	(* --- Visu controler --- *)
	iMAX_AXIS_FRAMES						: USINT := 20;														(* Maximum frames of displayed axis in manual mode *)
	iMAX_CYLINDER_FRAMES					: USINT := 42;														(* Maximum frames of displayed cylinders in manual mode *)
	iMAX_OUTPUT_FRAMES						: USINT := 144;														(* Maximum frames of displayed outputs in manual mode *)
	iMAX_INPUT_FRAMES						: USINT := 144;														(* Maximum frames of displayed inputs in manual mode *)
	iMAX_SAFE_INPUT_FRAMES					: USINT := 36;														(* Maximum frames of displayed safe inputs in manual mode *)
	iMAX_SAFE_OUTPUT_FRAMES					: USINT := 36;														(* Maximum frames of displayed safe outputs in manual mode *)
	iMAX_ROBOT_FRAMES						: USINT := 10;														(* Maximum frames of displayed safe outputs in manual mode *)
	                                                        													
	iAXIS_PER_PAGE							: USINT := 2;														(* Number of axis displayed on single page *)
	iCYLINDERS_PER_PAGE						: USINT := 3;														(* Number of cylinders dislayed on single page *)
	iOUTPUTS_PER_PAGE						: USINT := 12;														(* Number of outputs displayed on single page *)
	iINPUTS_PER_PAGE						: USINT := 12;														(* Number of inputs displayed on single page *)
	iSAFE_INPUTS_PER_PAGE					: USINT := 6;														(* Number of safe inputs displayed on single page*)
	iSAFE_OUTPUTS_PER_PAGE					: USINT := 6;														(* Number of safe outputs displayed on single page *)
	iRECIPE_PARAMETERS_PER_PAGE				: USINT := 8;														(* Number of recipes parameters displayed on single page *)
	iROBOTS_PER_PAGE						: USINT := 1;														(* Number of recipes parameters displayed on single page *)
	
	iMAX_AXIS_PAGES							: USINT := iMAX_AXIS_FRAMES / iAXIS_PER_PAGE;						(* Defines maximum pages of axis HMI frames in manual mode *)
	iMAX_CYLINDER_PAGES						: USINT := iMAX_CYLINDER_FRAMES / iCYLINDERS_PER_PAGE;				(* Defines maximum pages of cylinders HMI frames in manual mode *)
	iMAX_OUTPUT_PAGES						: USINT := iMAX_OUTPUT_FRAMES / iOUTPUTS_PER_PAGE;					(* Defines maximum pages of digital outputs HMI frames in manual mode *)
	iMAX_INPUT_PAGES						: USINT := iMAX_INPUT_FRAMES / iINPUTS_PER_PAGE;					(* Defines maximum pages of digital inputs HMI frames in manual mode *)
	iMAX_SAFE_INPUT_PAGES					: USINT := iMAX_SAFE_INPUT_FRAMES / iSAFE_INPUTS_PER_PAGE;			(* Defines maximum pages of safe inputs HMI frames in manual mode *)
	iMAX_SAFE_OUTPUT_PAGES					: USINT := iMAX_SAFE_OUTPUT_FRAMES / iSAFE_OUTPUTS_PER_PAGE;		(* Defines maximum pages of safe outputs HMI frames in manual mode *)
	iMAX_RECIPES_PAGES						: USINT := iMAX_NUMBER_OF_RECIPES / iRECIPE_PARAMETERS_PER_PAGE;	(* Defines maximum pages of recipes parameter HMI frames in manual mode *)
	iMAX_ROBOT_PAGES						: USINT := iMAX_ROBOT_FRAMES / iROBOTS_PER_PAGE;					(* Defines maximum pages of robots HMI frames *)

	(* --- CSV Data Exchanger --- *)
	iMAX_CSV_ROWS 							: UDINT := 100;
	iMAX_CSV_COLUMNS 						: UDINT := 8;
	iMAX_CSV_FIELD_LENGTH					: UDINT := 100;
END_VAR
VAR_GLOBAL
	(* --- Machine data ---*)
	sMACHINE_NAME							: STRING := 'PSE Shell Test Machine';								(* Full machine project name *)
	sSOFTWARE_VERSION						: STRING := '1.0.1.0';												(* Last taged version of control software *)
	
	(* --- Shell common features ---*)
	fbMachineTime							: FB_LocalSystemTime; 												(* Main machine clock - used by implementation of other utilites like Logger and Alarm Controler *)
	fbMachineLogger 						: FB_FileLogger; 													(* Main machine logger - registers everything that happens on machine *)

	(* --- Shell Machine ---*)
	stShell : ST_Shell;	(* This structure contains references to Shell modules, recipe parameters and auxilary bit flags *)
END_VAR

// ---- POUs/Libs/0_Checks/GVL_Checks.TcGVL
{attribute 'qualified_only'}
VAR_GLOBAL PERSISTENT
	dCheckBounds					: DINT;			// Licznik przekroczen zakresu indexow, np. tablic
	dCheckDivDInt					: DINT;			// Licznik prob dzielenia Dint przez 0
	dCheckDivLInt					: DINT; 		// Licznik prob dzielenia LInt przez 0
	dCheckDivLReal					: DINT; 		// Licznik prob dzielenia LREAL przez 0
	dCheckDivReal					: DINT; 		// Licznik prob dzielenia REAL przez 0
	dCheckRangeSigned				: DINT;			// Licznik przekroczen liczby znakowej
	dCheckRangeUnsigned				: DINT; 		// Licznik przekroczen liczby bezznakowej
END_VAR

// ---- POUs/Libs/Alarms/AlarmControler/I_AlarmControler.TcIO
INTERFACE I_AlarmControler

PROPERTY Active : REFERENCE TO BOOL
GET
END_GET
END_PROPERTY

PROPERTY ActiveCritical : REFERENCE TO UDINT
GET
END_GET
END_PROPERTY

PROPERTY ActiveError : REFERENCE TO UDINT
GET
END_GET
END_PROPERTY

PROPERTY ActiveInfo : REFERENCE TO UDINT
GET
END_GET
END_PROPERTY

PROPERTY ActiveVerbose : REFERENCE TO UDINT
GET
END_GET
END_PROPERTY

PROPERTY ActiveWarrning : REFERENCE TO UDINT
GET
END_GET
END_PROPERTY

PROPERTY Busy : REFERENCE TO BOOL
GET
END_GET
END_PROPERTY

PROPERTY Error : REFERENCE TO BOOL
GET
END_GET
END_PROPERTY

PROPERTY FileName : STRING
GET
END_GET
SET
END_SET
END_PROPERTY

PROPERTY MaxEvents : UDINT
GET
END_GET
END_PROPERTY

METHOD MR_Abort : BOOL
VAR_INPUT
END_VAR
END_METHOD

METHOD MR_Clear : BOOL
VAR_INPUT
	ipFilter : I_TcEventFilter;
	bResetConfirmation : BOOL;
END_VAR
END_METHOD

METHOD MR_ClearAll : BOOL
VAR_INPUT
	bResetConfirmation : BOOL;
END_VAR
END_METHOD

METHOD MR_Confirm : BOOL
VAR_INPUT
	ipFilter : I_TcEventFilter;
END_VAR
END_METHOD

METHOD MR_ConfirmAll : BOOL
VAR_INPUT
	bResetConfirmation : BOOL;
END_VAR
END_METHOD

METHOD MR_Export : BOOL
VAR_INPUT
END_VAR
END_METHOD

METHOD MR_FirstCycle : BOOL
VAR_INPUT
	sName 		: STRING;
	sFileName 	: STRING;
END_VAR
END_METHOD

METHOD MR_Init : BOOL
VAR_INPUT
END_VAR
END_METHOD

PROPERTY Name : REFERENCE TO STRING
GET
END_GET
END_PROPERTY

PROPERTY State : REFERENCE TO E_AlarmControlerState
GET
END_GET
END_PROPERTY

END_INTERFACE

// ---- POUs/Libs/Axis/I_UniversalAxis.TcIO
INTERFACE I_UniversalAxis

PROPERTY Acceleration : LREAL
GET
END_GET
SET
END_SET
END_PROPERTY

PROPERTY Active : REFERENCE TO BOOL
GET
END_GET
END_PROPERTY

PROPERTY ActualPosition : REFERENCE TO LREAL
GET
END_GET
END_PROPERTY

PROPERTY ActualVelocity : REFERENCE TO LREAL
GET
END_GET
END_PROPERTY

PROPERTY AxisErrorID : REFERENCE TO UDINT
GET
END_GET
END_PROPERTY

PROPERTY AxisRef : AXIS_REF
GET
END_GET
SET
END_SET
END_PROPERTY

PROPERTY BufferMode : MC_BufferMode
GET
END_GET
SET
END_SET
END_PROPERTY

PROPERTY Busy : REFERENCE TO BOOL
GET
END_GET
END_PROPERTY

PROPERTY Deceleration : LREAL
GET
END_GET
SET
END_SET
END_PROPERTY

PROPERTY Direction : Tc2_MC2.MC_Direction
GET
END_GET
SET
END_SET
END_PROPERTY

PROPERTY Error : REFERENCE TO BOOL
GET
END_GET
END_PROPERTY

PROPERTY ErrorID : REFERENCE TO UDINT
GET
END_GET
END_PROPERTY

PROPERTY Halted : REFERENCE TO BOOL
GET
END_GET
END_PROPERTY

PROPERTY InPosition : REFERENCE TO BOOL
GET
END_GET
END_PROPERTY

PROPERTY InVelocity : REFERENCE TO BOOL
GET
END_GET
END_PROPERTY

PROPERTY IsHomed : REFERENCE TO BOOL
GET
END_GET
END_PROPERTY

PROPERTY Jerk : LREAL
GET
END_GET
SET
END_SET
END_PROPERTY

PROPERTY JogAcceleration : LREAL
GET
END_GET
SET
END_SET
END_PROPERTY

PROPERTY JogDeceleration : LREAL
GET
END_GET
SET
END_SET
END_PROPERTY

PROPERTY JogDirection : E_AxisJogDirection
GET
END_GET
SET
END_SET
END_PROPERTY

PROPERTY JogDone : REFERENCE TO BOOL
GET
END_GET
END_PROPERTY

PROPERTY JogJerk : LREAL
GET
END_GET
SET
END_SET
END_PROPERTY

PROPERTY JogMode : E_JogMode
GET
END_GET
SET
END_SET
END_PROPERTY

PROPERTY JogPosition : LREAL
GET
END_GET
SET
END_SET
END_PROPERTY

PROPERTY JogVelocity : LREAL
GET
END_GET
SET
END_SET
END_PROPERTY

PROPERTY LagError : LREAL
GET
END_GET
END_PROPERTY

PROPERTY MoveActive : REFERENCE TO BOOL
GET
END_GET
END_PROPERTY

METHOD MR_Abort : BOOL
END_METHOD

METHOD MR_FirstCycle
VAR_INPUT
	sName 				: STRING; 	(* Axis object name *)
	sMeasurementUnits	: STRING;	(* Measurement units used by axis *)
	bModulo				: BOOL;		(* Axis is periodic *)
END_VAR
END_METHOD

METHOD MR_Halt : BOOL
END_METHOD

METHOD MR_Home : BOOL
VAR_INPUT
	lrHomePosition : LREAL;
END_VAR
END_METHOD

METHOD MR_Init : BOOL
END_METHOD

METHOD MR_Jog : BOOL
VAR_INPUT
	//lrJogPosition : LREAL;
	//eJogDirection : E_AxisJogDirection;
	//eJogMode	  : E_JogMode;
	bJogActive	  : BOOL;
END_VAR
END_METHOD

METHOD MR_MoveAbsolute : BOOL
VAR_INPUT
	lrAbsolutePosition : LREAL;
END_VAR
END_METHOD

METHOD MR_MoveAdditive : BOOL
VAR_INPUT
	lrRelativeDistance : LREAL;
END_VAR
END_METHOD

METHOD MR_MoveRelative : BOOL
VAR_INPUT
	lrRelativeDistance : LREAL;
END_VAR
END_METHOD

METHOD MR_MoveVelocity : BOOL
END_METHOD

METHOD MR_Reset : BOOL
END_METHOD

METHOD MR_Stop : BOOL
END_METHOD

PROPERTY Name : STRING
GET
END_GET
SET
END_SET
END_PROPERTY

PROPERTY Options : ST_MoveOptions
GET
END_GET
SET
END_SET
END_PROPERTY

PROPERTY Override : LREAL
GET
END_GET
SET
END_SET
END_PROPERTY

PROPERTY PowerOn : REFERENCE TO BOOL
GET
END_GET
END_PROPERTY

PROPERTY SetpointPosition : LREAL
GET
END_GET
END_PROPERTY

PROPERTY SetpointVelocity : LREAL
GET
END_GET
END_PROPERTY

PROPERTY State : REFERENCE TO E_AxisState
GET
END_GET
END_PROPERTY

PROPERTY StatePlcOpen : REFERENCE TO E_AxisStatePlcOpen
GET
END_GET
END_PROPERTY

PROPERTY StopDeceleration : LREAL
GET
END_GET
SET
END_SET
END_PROPERTY

PROPERTY StopJerk : LREAL
GET
END_GET
SET
END_SET
END_PROPERTY

PROPERTY Stopped : REFERENCE TO BOOL
GET
END_GET
END_PROPERTY

PROPERTY Unit : STRING
GET
END_GET
SET
END_SET
END_PROPERTY

PROPERTY Velocity : LREAL
GET
END_GET
SET
END_SET
END_PROPERTY

END_INTERFACE

// ---- POUs/Libs/Communication/TcpIp/Tcp Device/I_TcpDevice.TcIO
INTERFACE I_TcpDevice

PROPERTY Active : REFERENCE TO BOOL
GET
END_GET
END_PROPERTY

PROPERTY AmsNetId : T_IPv4Addr
GET
END_GET
SET
END_SET
END_PROPERTY

PROPERTY Error : REFERENCE TO BOOL
GET
END_GET
END_PROPERTY

PROPERTY ErrorID : REFERENCE TO UDINT
GET
END_GET
END_PROPERTY

PROPERTY Host : T_IPv4Addr
GET
END_GET
SET
END_SET
END_PROPERTY

PROPERTY LastRecivedMessage : ST_TcpBufferData
GET
END_GET
END_PROPERTY

METHOD MR_Abort : BOOL
VAR_INPUT
END_VAR
END_METHOD

METHOD MR_FirstCycle : BOOL
VAR_INPUT
	sName 		: STRING;		(*  *)
	sHost		: T_IPv4Addr;	(*  *)
	sAmsNetID	: T_AmsNetID;	(*  *)
	iPort		: UINT;			(*  *)
	tTimeout	: TIME;			(*  *)
END_VAR
END_METHOD

METHOD MR_Init : BOOL
VAR_INPUT
END_VAR
END_METHOD

PROPERTY NextRecivedMessage : ST_TcpBufferData
GET
END_GET
END_PROPERTY

PROPERTY Port : UINT
GET
END_GET
SET
END_SET
END_PROPERTY

PROPERTY State : REFERENCE TO E_TcpIpDeviceState
GET
END_GET
END_PROPERTY

PROPERTY Timeout : TIME
GET
END_GET
SET
END_SET
END_PROPERTY

END_INTERFACE

// ---- POUs/Libs/Cylinder/Universal Cylinder/I_UniversalCylinder.TcIO
INTERFACE I_UniversalCylinder

PROPERTY Active : REFERENCE TO BOOL
GET
END_GET
END_PROPERTY

PROPERTY ActiveTimeout : TIME
GET
END_GET
SET
END_SET
END_PROPERTY

PROPERTY Busy : REFERENCE TO BOOL
GET
END_GET
END_PROPERTY

PROPERTY Delay : TIME
GET
END_GET
SET
END_SET
END_PROPERTY

PROPERTY Error : REFERENCE TO BOOL
GET
END_GET
END_PROPERTY

PROPERTY ErrorID : REFERENCE TO E_CylinderError
GET
END_GET
END_PROPERTY

PROPERTY HomeTimeout : TIME
GET
END_GET
SET
END_SET
END_PROPERTY

PROPERTY MoveActiveTime : REFERENCE TO TIME
GET
END_GET
END_PROPERTY

PROPERTY MoveHomeTime : REFERENCE TO TIME
GET
END_GET
END_PROPERTY

METHOD MR_Abort : BOOL
VAR_INPUT
END_VAR
END_METHOD

METHOD MR_FirstCycle : BOOL
VAR_INPUT
sName 							: STRING;
	sHomeSensorModuleType			: STRING;
	sHomeSensorPortID				: STRING;
	sActiveSensorModuleType			: STRING;
	sActiveSensorPortID				: STRING;
	tGoHomeTimeout					: TIME;
	tGoActiveTimeout				: TIME;
	tDelay							: TIME;
END_VAR
END_METHOD

METHOD MR_GoActive : BOOL
VAR_INPUT
END_VAR
END_METHOD

METHOD MR_GoHome : BOOL
VAR_INPUT
END_VAR
END_METHOD

METHOD MR_Init : BOOL
VAR_INPUT
END_VAR
END_METHOD

METHOD MR_Release : BOOL
VAR_INPUT
END_VAR
END_METHOD

METHOD MR_Reset : BOOL
VAR_INPUT
END_VAR
END_METHOD

PROPERTY Name : STRING
GET
END_GET
SET
END_SET
END_PROPERTY

PROPERTY PositionActive : REFERENCE TO BOOL
GET
END_GET
END_PROPERTY

PROPERTY PositionHold : REFERENCE TO BOOL
GET
END_GET
END_PROPERTY

PROPERTY PositionHome : REFERENCE TO BOOL
GET
END_GET
END_PROPERTY

PROPERTY Simulation : BOOL
GET
END_GET
SET
END_SET
END_PROPERTY

PROPERTY State : REFERENCE TO E_CylinderState
GET
END_GET
END_PROPERTY

END_INTERFACE

// ---- POUs/Libs/Digital Devices/Digital Device/I_DigitalDevice.TcIO
INTERFACE I_DigitalDevice

PROPERTY ModuleType : REFERENCE TO STRING
GET
END_GET
END_PROPERTY

METHOD MR_FirstCycle : BOOL
VAR_INPUT
	sName 			: STRING;
	sModuleType 	: STRING;
	sPortID			: STRING;
END_VAR
END_METHOD

PROPERTY Name : REFERENCE TO STRING
GET
END_GET
END_PROPERTY

PROPERTY PortID : REFERENCE TO STRING
GET
END_GET
END_PROPERTY

END_INTERFACE

// ---- POUs/Libs/Digital Devices/Digital Input/I_DigitalInput.TcIO
INTERFACE I_DigitalInput EXTENDS I_DigitalDevice

PROPERTY EnableForce : BOOL
GET
END_GET
SET
END_SET
END_PROPERTY

PROPERTY FallingTrigger : BOOL
GET
END_GET
END_PROPERTY

PROPERTY In : BOOL
GET
END_GET
END_PROPERTY

METHOD MR_ResetForceValue
END_METHOD

METHOD MR_SetForceValue
END_METHOD

PROPERTY RisingTrigger : BOOL
GET
END_GET
END_PROPERTY

END_INTERFACE

// ---- POUs/Libs/Digital Devices/Digital Output/I_DigitalOutput.TcIO
INTERFACE I_DigitalOutput EXTENDS I_DigitalDevice

PROPERTY Out : BOOL
GET
END_GET
SET
END_SET
END_PROPERTY

END_INTERFACE

// ---- POUs/Libs/Digital Devices/Lamp Indicator/I_Lamp.TcIO
INTERFACE I_Lamp EXTENDS I_DigitalDevice

METHOD MR_LampBlink : BOOL
VAR_INPUT
	tBlinkTime : TIME;
END_VAR
END_METHOD

METHOD MR_LampOff : BOOL
VAR_INPUT
END_VAR
END_METHOD

METHOD MR_LampOn : BOOL
VAR_INPUT
END_VAR
END_METHOD

PROPERTY Status : REFERENCE TO E_LampState
GET
END_GET
END_PROPERTY

END_INTERFACE

// ---- POUs/Libs/Fixtures/I_UniversalFixture.TcIO
INTERFACE I_UniversalFixture

PROPERTY Active : REFERENCE TO BOOL
GET
END_GET
END_PROPERTY

PROPERTY Busy : REFERENCE TO BOOL
GET
END_GET
END_PROPERTY

PROPERTY Error : REFERENCE TO BOOL
GET
END_GET
END_PROPERTY

METHOD MR_Abort : BOOL
VAR_INPUT
END_VAR
END_METHOD

METHOD MR_Close : BOOL
VAR_INPUT
END_VAR
END_METHOD

METHOD MR_FirstCycle : BOOL
VAR_INPUT
	sFixtureName 		: STRING;		(*  *)
	sHost				: T_IPv4Addr;	(*  *)
	sAmsNetID 			: T_AmsNetID;	(*  *)
	iPort				: UINT;			(*  *)
	tTimeout			: TIME;			(*  *)
	bUseLogger			: BOOL;			(*  *)
	bClientConnection 	: BOOL;			(*  *)
	sFileDir			: STRING;		(*  *)
	sFileName			: STRING;		(*  *)
	bCreateFileAtStart	: BOOL;
	bAddHeader			: BOOL;
	bAddTimeStamp		: BOOL;	
END_VAR
END_METHOD

METHOD MR_Init : BOOL
END_METHOD

METHOD MR_Measure : BOOL
VAR_INPUT
	iSampleID : UINT;
END_VAR
END_METHOD

METHOD MR_Open : BOOL
VAR_INPUT
END_VAR
END_METHOD

METHOD MR_Reset : BOOL
VAR_INPUT
END_VAR
END_METHOD

PROPERTY RecivedUtuData : REFERENCE TO STRING
GET
END_GET
END_PROPERTY

PROPERTY ref_MeasurementLogger : REFERENCE TO FB_TXTDataExchanger
GET
END_GET
END_PROPERTY

PROPERTY ref_TcpClient : REFERENCE TO FB_TcpClient
GET
END_GET
END_PROPERTY

PROPERTY ref_TcpServer : REFERENCE TO FB_TcpServer
GET
END_GET
END_PROPERTY

PROPERTY SampleID : REFERENCE TO UDINT
GET
END_GET
END_PROPERTY

PROPERTY SampleResult : REFERENCE TO E_UniversalFixtureSampleResult
GET
END_GET
END_PROPERTY

PROPERTY ABSTRACT SocketOpen : REFERENCE TO BOOL
GET
END_GET
END_PROPERTY

PROPERTY State : REFERENCE TO E_UniversalFixtureState
GET
END_GET
END_PROPERTY

END_INTERFACE

// ---- POUs/Libs/Platform/Universal Machine/I_UniversalMachine.TcIO
INTERFACE I_UniversalMachine

PROPERTY Active : REFERENCE TO BOOL
GET
END_GET
END_PROPERTY

PROPERTY Error : REFERENCE TO BOOL
GET
END_GET
END_PROPERTY

METHOD MR_Abort : BOOL
VAR_INPUT
END_VAR
END_METHOD

METHOD MR_Init : BOOL
VAR_INPUT
END_VAR
END_METHOD

METHOD MR_Reset : BOOL
VAR_INPUT
END_VAR
END_METHOD

METHOD MR_Start : BOOL
VAR_INPUT
END_VAR
END_METHOD

METHOD MR_Stop : BOOL
VAR_INPUT
END_VAR
END_METHOD

METHOD MR_SwitchToAuto : BOOL
VAR_INPUT
END_VAR
END_METHOD

METHOD MR_SwitchToManual : BOOL
VAR_INPUT
END_VAR
END_METHOD

PROPERTY Running : REFERENCE TO BOOL
GET
END_GET
END_PROPERTY

PROPERTY State : REFERENCE TO E_MachineCtrlState
GET
END_GET
END_PROPERTY

END_INTERFACE

// ---- POUs/Libs/Platform/Universal Safety/I_UniversalSafety.TcIO
INTERFACE I_UniversalSafety

METHOD MR_Abort : BOOL
VAR_INPUT
END_VAR
END_METHOD

METHOD MR_FirstCycle : BOOL
VAR_INPUT
END_VAR
END_METHOD

METHOD MR_Init : BOOL
VAR_INPUT
END_VAR
END_METHOD

METHOD MR_Reset : BOOL
VAR_INPUT
END_VAR
END_METHOD

END_INTERFACE

// ---- POUs/Libs/Robots/Mitsubishi/I_CR800EtherCAT.TcIO
INTERFACE I_CR800EtherCAT

PROPERTY ActionNumber : UINT
GET
END_GET
SET
END_SET
END_PROPERTY

PROPERTY Active : REFERENCE TO BOOL
GET
END_GET
END_PROPERTY

PROPERTY AutoModeStarted : REFERENCE TO BOOL
GET
END_GET
END_PROPERTY

PROPERTY BatteryLow : BOOL
GET
END_GET
END_PROPERTY

PROPERTY BatteryReset : BOOL
GET
END_GET
SET
END_SET
END_PROPERTY

PROPERTY BatteryResetCompleted : BOOL
GET
END_GET
END_PROPERTY

PROPERTY Busy : REFERENCE TO BOOL
GET
END_GET
END_PROPERTY

PROPERTY CR800PoweredOn : BOOL
GET
END_GET
END_PROPERTY

PROPERTY CycleStop : BOOL
GET
END_GET
SET
END_SET
END_PROPERTY

PROPERTY CycleStopping : BOOL
GET
END_GET
END_PROPERTY

PROPERTY DoingAction : REFERENCE TO BOOL
GET
END_GET
END_PROPERTY

PROPERTY EmergencyStopOccuring : BOOL
GET
END_GET
END_PROPERTY

PROPERTY Error : REFERENCE TO BOOL
GET
END_GET
END_PROPERTY

PROPERTY ErrorName : STRING
GET
END_GET
END_PROPERTY

PROPERTY ErrorOccuring : BOOL
GET
END_GET
END_PROPERTY

PROPERTY ErrorReset : BOOL
GET
END_GET
SET
END_SET
END_PROPERTY

PROPERTY EthercatData : REFERENCE TO ST_CR800EthercatData
GET
END_GET
END_PROPERTY

PROPERTY InAutomaticMode : BOOL
GET
END_GET
END_PROPERTY

PROPERTY InRemoteMode : BOOL
GET
END_GET
END_PROPERTY

PROPERTY InTeachingMode : BOOL
GET
END_GET
END_PROPERTY

PROPERTY IsHomed : REFERENCE TO BOOL
GET
END_GET
END_PROPERTY

METHOD  MR_Abort : BOOL
END_METHOD

METHOD MR_BatteryReset : BOOL
END_METHOD

METHOD MR_CyclePause : BOOL
END_METHOD

METHOD MR_CycleStop : BOOL
END_METHOD

METHOD MR_DoAction : BOOL
VAR_INPUT
	iActionNumber : UINT ;
END_VAR
END_METHOD

METHOD MR_GoAuto : BOOL
END_METHOD

METHOD MR_GoHome : BOOL
END_METHOD

METHOD MR_Init : BOOL
END_METHOD

METHOD MR_Reset : BOOL
END_METHOD

METHOD MR_ResetCR800Err : BOOL
END_METHOD

METHOD MR_RestoreAuto : BOOL
END_METHOD

METHOD MR_RestoreCycle : BOOL
END_METHOD

METHOD MR_SendPosition1 : BOOL 
VAR_INPUT
	lrPositionX1	: LREAL;
	lrPositionY1	: LREAL;
	lrRotation1		: LREAL;
END_VAR
END_METHOD

METHOD MR_SendPosition2 : BOOL 
VAR_INPUT
	lrPositionX2	: LREAL;
	lrPositionY2	: LREAL;
	lrRotation2		: LREAL;
END_VAR
END_METHOD

METHOD MR_UpdateRecipies : BOOL
END_METHOD

PROPERTY Name : STRING
GET
END_GET
SET
END_SET
END_PROPERTY

PROPERTY OperationRightsEnable : BOOL
GET
END_GET
SET
END_SET
END_PROPERTY

PROPERTY OperationRightsEnabled : BOOL
GET
END_GET
END_PROPERTY

PROPERTY Override : USINT
GET
END_GET
SET
END_SET
END_PROPERTY

PROPERTY Pausing : BOOL
GET
END_GET
END_PROPERTY

PROPERTY PUBLIC ProgramOperating : BOOL
GET
END_GET
END_PROPERTY

PROPERTY ProgramReset : BOOL
GET
END_GET
SET
END_SET
END_PROPERTY

PROPERTY ProgramSelectionEnabled : BOOL
GET
END_GET
END_PROPERTY

PROPERTY ProgramStart : BOOL
GET
END_GET
SET
END_SET
END_PROPERTY

PROPERTY ProgramStop2 : BOOL
GET
END_GET
SET
END_SET
END_PROPERTY

PROPERTY PUBLIC ProgramStopped : BOOL
GET
END_GET
END_PROPERTY

PROPERTY RequestNumber : UINT
GET
END_GET
SET
END_SET
END_PROPERTY

PROPERTY SendingPosition1 : REFERENCE TO BOOL
GET
END_GET
END_PROPERTY

PROPERTY SendingPosition2 : REFERENCE TO BOOL
GET
END_GET
END_PROPERTY

PROPERTY ServoIsOff : BOOL
GET
END_GET
END_PROPERTY

PROPERTY ServoIsOn : BOOL
GET
END_GET
END_PROPERTY

PROPERTY ServoOff : BOOL
GET
END_GET
SET
END_SET
END_PROPERTY

PROPERTY ServoOn : BOOL
GET
END_GET
SET
END_SET
END_PROPERTY

PROPERTY State : REFERENCE TO E_CR800State
GET
END_GET
END_PROPERTY

PROPERTY StopSTS : BOOL
GET
END_GET
END_PROPERTY

PROPERTY Uninitialized : REFERENCE TO BOOL
GET
END_GET
END_PROPERTY

PROPERTY UserDefinedArea1 : BOOL
GET
END_GET
END_PROPERTY

PROPERTY UserDefinedArea2 : BOOL
GET
END_GET
END_PROPERTY

PROPERTY UserDefinedArea3 : BOOL
GET
END_GET
END_PROPERTY

PROPERTY UserDefinedArea4 : BOOL
GET
END_GET
END_PROPERTY

PROPERTY UserDefinedArea5 : BOOL
GET
END_GET
END_PROPERTY

PROPERTY UserDefinedArea6 : BOOL
GET
END_GET
END_PROPERTY

PROPERTY UserDefinedArea7 : BOOL
GET
END_GET
END_PROPERTY

PROPERTY UserDefinedArea8 : BOOL
GET
END_GET
END_PROPERTY

END_INTERFACE

// ---- POUs/Libs/Utilities/Beckhoff UPS/CX5xxx/I_BeckhoffUpsCX5xxx.TcIO
INTERFACE I_BeckhoffUpsCX5xxx EXTENDS I_UniversalCxUps

PROPERTY PersistentMode : E_PersistentMode
GET
END_GET
SET
END_SET
END_PROPERTY

PROPERTY RecoverTime : Time
GET
END_GET
SET
END_SET
END_PROPERTY

PROPERTY UpsMode : E_S_UPS_Mode
GET
END_GET
SET
END_SET
END_PROPERTY

PROPERTY UpsPort : UINT
GET
END_GET
SET
END_SET
END_PROPERTY

END_INTERFACE

// ---- POUs/Libs/Utilities/Beckhoff UPS/Universal CX/I_UniversalCxUps.TcIO
INTERFACE I_UniversalCxUps

METHOD MR_FirstCycle : BOOL
VAR_INPUT
	sName 		: STRING;
	sNetID		: STRING;
	iPlcPort 	: UINT;
	tTimeout	: TIME;
END_VAR
END_METHOD

PROPERTY Name : STRING
GET
END_GET
SET
END_SET
END_PROPERTY

PROPERTY NetId : STRING
GET
END_GET
SET
END_SET
END_PROPERTY

PROPERTY PlcPort : UINT
GET
END_GET
SET
END_SET
END_PROPERTY

PROPERTY PowerOk : REFERENCE TO BOOL
GET
END_GET
END_PROPERTY

PROPERTY Timeout : Time
GET
END_GET
SET
END_SET
END_PROPERTY

END_INTERFACE

// ---- POUs/Libs/Utilities/CSV Data Exchanger/I_CSVDataExchanger.TcIO
INTERFACE I_CSVDataExchanger

PROPERTY Active : REFERENCE TO BOOL
GET
END_GET
END_PROPERTY

PROPERTY Busy : REFERENCE TO BOOL
GET
END_GET
END_PROPERTY

PROPERTY Error : REFERENCE TO BOOL
GET
END_GET
END_PROPERTY

PROPERTY ErrorID : REFERENCE TO UDINT
GET
END_GET
END_PROPERTY

METHOD MR_Abort : BOOL
END_METHOD

METHOD MR_FirstCycle : BOOL
VAR_INPUT
	sAmsNetId					: T_AmsNetId;	(* TwinCAT system network address *)
	sFileDir					: T_MaxString;	(* CSV source file path *)
	sFileName 					: T_MaxString;	(* CSV source file name *)
//	bCreateFile					: BOOL;			(* If true FB will create file under given path *)
//	bAddHeader					: BOOL;			(* If true there will be a header at the beginning of the doc *)
	(*	In USA/UK the CSV field separator is a comma.
	In Germany and some other European countries the CSV field separator is a semicolon. *)
	bChangeSeparatorToComma		: BOOL;
END_VAR
END_METHOD

METHOD MR_Init : BOOL
VAR_INPUT
END_VAR
END_METHOD

METHOD MR_Reset : BOOL
END_METHOD

METHOD MR_SelectAll : BOOL
VAR_INPUT
	iArrDataBaseAdr 		: PVOID; 		(* A pointer to the string array where the 100 records (max.) from CSV file table are stored *)
END_VAR
END_METHOD

METHOD MR_SelectPath : BOOL
VAR_INPUT
	sFileDir								: T_MaxString; 			(* CSV source file directory name *)
	sFileName 								: T_MaxString; 			(* CSV source file name *)
END_VAR
END_METHOD

METHOD MR_SelectRow : BOOL
VAR_INPUT
	iColumnToSearch 			: UDINT;		(* Column number to search the value in; columns are counted from 1 *)
	sValueToSearch				: STRING;		(* Value that you are looking for *)
	iArrParsedStringAdr 		: PVOID;		(* A pointer to the string array where the matched row with the search value is stored as a string array *)
END_VAR

VAR_OUTPUT
	sRowResult					: STRING;
END_VAR
END_METHOD

END_INTERFACE

// ---- POUs/Libs/Utilities/File Logger/I_FileLogger.TcIO
INTERFACE I_FileLogger

PROPERTY Active : REFERENCE TO BOOL
GET
END_GET
END_PROPERTY

PROPERTY Busy : REFERENCE TO BOOL
GET
END_GET
END_PROPERTY

PROPERTY Error : REFERENCE TO BOOL
GET
END_GET
END_PROPERTY

PROPERTY ErrorID : REFERENCE TO UDINT
GET
END_GET
END_PROPERTY

METHOD MR_Abort : BOOL
VAR_INPUT
END_VAR
END_METHOD

METHOD MR_AddLogs : BOOL
VAR_INPUT
	sLogMessage : STRING;
END_VAR
END_METHOD

METHOD MR_FirstCycle : BOOL
VAR_INPUT
	sName 		: STRING;
	sFileDir	: STRING(255);
	sFileName	: STRING(255);
	sAmsNetId	: T_AmsNetID;
	bAddTimeStamp	: BOOL;
	bAddHeader		: BOOL;
END_VAR
END_METHOD

METHOD MR_Init : BOOL
VAR_INPUT
END_VAR
END_METHOD

METHOD MR_Reset : BOOL
VAR_INPUT
END_VAR
END_METHOD

END_INTERFACE

// ---- POUs/Libs/Utilities/Recipes Manager/I_RecipeParameter.TcIO
INTERFACE I_RecipeParameter

PROPERTY BitValue : REFERENCE TO BOOL
GET
END_GET
END_PROPERTY

PROPERTY DataType : REFERENCE TO E_VisuCtrlRecipeParameterType
GET
END_GET
END_PROPERTY

PROPERTY FileValue : REFERENCE TO STRING
GET
END_GET
END_PROPERTY

PROPERTY IntValue : REFERENCE TO DINT
GET
END_GET
END_PROPERTY

PROPERTY Name : REFERENCE TO STRING
GET
END_GET
END_PROPERTY

PROPERTY RealValue : REFERENCE TO REAL
GET
END_GET
END_PROPERTY

PROPERTY StringValue : REFERENCE TO STRING
GET
END_GET
END_PROPERTY

END_INTERFACE

// ---- POUs/Libs/Utilities/Recipes Manager/I_RecipesManager.TcIO
INTERFACE I_RecipesManager

PROPERTY Active : REFERENCE TO BOOL
GET
END_GET
END_PROPERTY

PROPERTY Busy : REFERENCE TO BOOL
GET
END_GET
END_PROPERTY

PROPERTY Error : REFERENCE TO BOOL
GET
END_GET
END_PROPERTY

PROPERTY ErrorID : REFERENCE TO DWORD
GET
END_GET
END_PROPERTY

PROPERTY LastResult : REFERENCE TO E_RecipesManagerReturns
GET
END_GET
END_PROPERTY

METHOD MR_Abort : BOOL
VAR_INPUT
END_VAR
END_METHOD

METHOD MR_Backup : BOOL
VAR_INPUT
	sRecipesDefinition		: STRING;
	sRecipeName				: STRING;
	sBackupStoragePath		: STRING;
END_VAR
END_METHOD

METHOD MR_Create : BOOL
VAR_INPUT
	sRecipesDefinition : STRING;
	sRecipeName : STRING;
END_VAR
END_METHOD

METHOD MR_GetRecipesNames : BOOL
VAR_INPUT
	sRecipesDefinition : STRING;
END_VAR
END_METHOD

METHOD MR_GetVariablesNames : BOOL
VAR_INPUT
	sRecipesDefinition	: STRING;
	sRecipeName : STRING;
END_VAR
END_METHOD

METHOD MR_GetVariableValues : BOOL
VAR_INPUT
	sRecipesDefinition	: STRING;
	sRecipeName : STRING;
END_VAR
END_METHOD

METHOD MR_Init : BOOL
VAR_INPUT
END_VAR
END_METHOD

METHOD MR_Load : BOOL
VAR_INPUT
	sRecipesDefinition : STRING;
	sRecipeName : STRING;
END_VAR
END_METHOD

METHOD MR_LoadAndWritte : BOOL
VAR_INPUT
	sRecipesDefinition : STRING;
	sRecipeName : STRING;
END_VAR
END_METHOD

METHOD MR_Read : BOOL
VAR_INPUT
	sRecipesDefinition : STRING;
	sRecipeName : STRING;
END_VAR
END_METHOD

METHOD MR_ReadAndSave : BOOL
VAR_INPUT
	sRecipesDefinition : STRING;
	sRecipeName : STRING;
END_VAR
END_METHOD

METHOD MR_Reload : BOOL
VAR_INPUT
	sRecipeName : STRING;
	sRecipesDefinition : STRING;
END_VAR
END_METHOD

METHOD MR_ReloadExternal : BOOL
VAR_INPUT
	sRecipeName 			: STRING;
	sRecipesDefinition 		: STRING;
	sBackupStoragePath		: STRING;
END_VAR
END_METHOD

METHOD MR_Remove : BOOL
VAR_INPUT
	sRecipesDefinition : STRING;
	sRecipeName : STRING;
END_VAR
END_METHOD

METHOD MR_Restore : BOOL
VAR_INPUT
	sRecipesDefinition		: STRING;
	sRecipeName				: STRING;
	sBackupStoragePath		: STRING;
END_VAR
END_METHOD

METHOD MR_Save : BOOL
VAR_INPUT
	sRecipesDefinition : STRING;
	sRecipeName : STRING;
END_VAR
END_METHOD

METHOD MR_Writte : BOOL
VAR_INPUT
	sRecipesDefinition : STRING;
	sRecipeName : STRING;
END_VAR
END_METHOD

PROPERTY RecipeCount : REFERENCE TO USINT
GET
END_GET
END_PROPERTY

PROPERTY RecipesDefinition : REFERENCE TO STRING
GET
END_GET
END_PROPERTY

PROPERTY RecipesNames : REFERENCE TO ARRAY [0..iMAX_NUMBER_OF_RECIPES-1] OF STRING;
GET
END_GET
END_PROPERTY

PROPERTY RecipeValues : REFERENCE TO ARRAY [0..iMAX_NUMBER_OF_VARIABLES_IN_RECIPES-1] OF STRING
//PROPERTY RecipeValues : ARRAY [0..iMAX_NUMBER_OF_VARIABLES_IN_RECIPES-1] OF STRING(iMAX_RECIPE_NAME_LENGTH)
GET
END_GET
END_PROPERTY

PROPERTY RecipeValuesAdr : REFERENCE TO ARRAY [0..iMAX_NUMBER_OF_VARIABLES_IN_RECIPES-1] OF PVOID
GET
END_GET
END_PROPERTY

PROPERTY State : REFERENCE TO E_RecipesManagerState
GET
END_GET
END_PROPERTY

END_INTERFACE

// ---- POUs/Libs/Utilities/TXT Data Exchanger/I_TXTDataExchanger.TcIO
INTERFACE I_TXTDataExchanger

PROPERTY Active : REFERENCE TO BOOL
GET
END_GET
END_PROPERTY

PROPERTY AmsNetId : STRING
GET
END_GET
SET
END_SET
END_PROPERTY

PROPERTY Busy : REFERENCE TO BOOL
GET
END_GET
END_PROPERTY

PROPERTY Error : REFERENCE TO BOOL
GET
END_GET
END_PROPERTY

PROPERTY ErrorID : REFERENCE TO UDINT
GET
END_GET
END_PROPERTY

PROPERTY FileDir : STRING
GET
END_GET
SET
END_SET
END_PROPERTY

PROPERTY FileName : STRING
GET
END_GET
SET
END_SET
END_PROPERTY

METHOD MR_Abort : BOOL
END_METHOD

METHOD MR_AddMESCommand : BOOL
VAR_INPUT
	sMachineID		: STRING;
	sOperatorID		: STRING;
	sPO				: STRING;
	sProductItem	: STRING;
	bLogOn			: BOOL;
END_VAR
END_METHOD

METHOD MR_Init : BOOL
VAR_INPUT
END_VAR
END_METHOD

METHOD MR_Reset : BOOL
END_METHOD

METHOD MR_SearchForFile : BOOL
VAR_INPUT
	sSearchFileName		: STRING;			(* Whole name of the search file (e.g.: "DemoFile.txt" *)
END_VAR

VAR_OUTPUT
	bFileFound	: BOOL;
END_VAR
END_METHOD

METHOD MR_SelectPath : BOOL
VAR_INPUT
	sFileDir								: STRING; 			(* CSV source file directory name *)
	sFileName 								: STRING; 			(* CSV source file name *)
END_VAR
END_METHOD

PROPERTY Name : STRING
GET
END_GET
SET
END_SET
END_PROPERTY

END_INTERFACE

// ---- POUs/Libs/Vision/Cognex/I_CognexCamera.TcIO
INTERFACE I_CognexCamera

PROPERTY Active : REFERENCE TO BOOL
GET
END_GET
END_PROPERTY

PROPERTY Busy : REFERENCE TO BOOL
GET
END_GET
END_PROPERTY

PROPERTY Error : REFERENCE TO BOOL
GET
END_GET
END_PROPERTY

PROPERTY ErrorID : REFERENCE TO UDINT
GET
END_GET
END_PROPERTY

METHOD MR_Abort : BOOL
VAR_INPUT
END_VAR
END_METHOD

METHOD MR_GetConnections : BOOL
END_METHOD

METHOD MR_GetExpr : BOOL
VAR_INPUT
	sCellIndexExpr	: STRING;
	iColumnExpr	: INT;
	iRowExpr	: INT;
END_VAR
END_METHOD

METHOD MR_GetFile : BOOL
END_METHOD

METHOD MR_GetFileList : BOOL
END_METHOD

METHOD MR_GetJob : BOOL
END_METHOD

METHOD MR_GetOnline : BOOL
END_METHOD

METHOD MR_GetPosition : BOOL
VAR_INPUT
	sPositionXVariable		: STRING;
	sPositionYVariable		: STRING;
	sRotationVariable		: STRING;
END_VAR

VAR_OUTPUT
	lrPositionX				: LREAL;
	lrPositionY				: LREAL;
	lrRotation				: LREAL;
END_VAR
END_METHOD

METHOD MR_GetValueEasyBuilder : BOOL
VAR_INPUT
	sEasyBuilderValueName	: STRING;
END_VAR
END_METHOD

METHOD MR_GetValues : BOOL
VAR_INPUT
	sVariable1				: STRING;
	sVariable2				: STRING;
	sVariable3				: STRING;
	sVariable4				: STRING;
END_VAR

VAR_OUTPUT
	lrValue1				: LREAL;
	lrValue2				: LREAL;
	lrValue3				: LREAL;
	lrValue4				: LREAL;	
END_VAR
END_METHOD

METHOD MR_GetValueSpreadsheet : BOOL
VAR_INPUT
	iColumnValueSpreadsheet		: INT;
	iRowValueSpreadsheet		: INT;
END_VAR
END_METHOD

METHOD MR_ImageTrigger : BOOL
END_METHOD

METHOD MR_Init : BOOL
END_METHOD

METHOD MR_LoadFile : BOOL
VAR_INPUT
	sLoadFileName	: STRING;
END_VAR
END_METHOD

METHOD MR_PutLive : BOOL
VAR_INPUT
	bEnableLiveAcquisition : INT;
END_VAR
END_METHOD

METHOD MR_PutPortnum : BOOL
VAR_INPUT
	iPortNumber : INT;
END_VAR
END_METHOD

METHOD MR_PutTimeout : BOOL
VAR_INPUT
	iTimeout 	: INT;
END_VAR
END_METHOD

METHOD MR_PutUpdate : BOOL
VAR_INPUT
	iUpdateNumber 	: INT;
END_VAR
END_METHOD

METHOD MR_PutWatch : BOOL
VAR_INPUT
	iColumnPut 		: INT;
	iRowPut 		: INT;
	iOutputEnable	: INT;
END_VAR
END_METHOD

METHOD MR_Reset : BOOL
END_METHOD

METHOD MR_ResetSystem : BOOL
END_METHOD

METHOD MR_SetJob : BOOL
VAR_INPUT
	iJobNumber 		: INT;
END_VAR
END_METHOD

METHOD MR_SetOnline : BOOL
VAR_INPUT
	bSetCameraOnline	: INT;
END_VAR
END_METHOD

METHOD MR_StoreFile : BOOL
VAR_INPUT
	sStoreFileName 	: STRING;
END_VAR
END_METHOD

PROPERTY Name : STRING
GET
END_GET
SET
END_SET
END_PROPERTY

PROPERTY ref_TcpClient : REFERENCE TO FB_TcpClient
GET
END_GET
END_PROPERTY

END_INTERFACE

// ---- POUs/Machine/Machine Control/I_MachineControl.TcIO
INTERFACE I_MachineControl EXTENDS I_UniversalMachine

PROPERTY Robots : REFERENCE TO FB_CR800EtherCAT
GET
END_GET
END_PROPERTY

END_INTERFACE

// ---- POUs/Machine/Alarm Control/PRG_AlarmControl.TcPOU
PROGRAM PRG_AlarmControl
VAR CONSTANT
	sDEFAULT_NAME		: STRING := 'Alarm Controler Test';	
	sDEFAULT_FILE_PATH	: STRING := 'C:\TwinCAT\Tests\EventLogger\events.csv';
END_VAR
VAR
	bFirstCycle			: BOOL := TRUE;
	fbAlarmControler 	: FB_AlarmControler;
	
	bInit 				: BOOL;
	bAbort				: BOOL;
END_VAR

IF bFirstCycle THEN
	bFirstCycle := FALSE;
	
	fbAlarmControler.MR_FirstCycle( sName		:= sDEFAULT_NAME,
									sFileName	:= sDEFAULT_FILE_PATH);
									
	(* Assign machine controler reference to Shell API*)
	stShell.stPlatform.ref_fbAlarmControler REF= fbAlarmControler;
	
	(* Set assignamnet done bit for visu controler *)
	stShell.stFlags.bAlarmCtrlAssignamentsDone := TRUE;
END_IF

fbAlarmControler();

END_PROGRAM

// ---- POUs/Libs/Alarms/AlarmControler/FB_AlarmControler.TcPOU
FUNCTION_BLOCK FB_AlarmControler EXTENDS FB_VisuEventsHandling IMPLEMENTS I_AlarmControler
VAR
	sName 					: STRING;					(*  *)

	bInit 					: BOOL;						(*  *)
	bAbort 					: BOOL;						(*  *)
	bClear					: BOOL;						(*  *)
	bClearAll 				: BOOL;						(*  *)
	bConfirm 				: BOOL;						(*  *)
	bConfirmAll 			: BOOL;						(*  *)
	bExport 				: BOOL;						(*  *)
	
	bResetConfirmation 		: BOOL;						(*  *)
	sFileName				: STRING;					(*  *)
	
	bActive 				: BOOL;						(*  *)
	bBusy					: BOOL;						(*  *)
	bError					: BOOL;						(*  *)
	iErrorID 				: HRESULT;					(*  *)
	iResult					: HRESULT;					(*  *)
	eAlarmControlerState 	: E_AlarmControlerState;	(*  *)
	
	ipFilter 				: I_TcEventFilter;			(*  *)
	fbEventLogger 			: FB_TcEventLogger;			(*  *)
END_VAR

(* Execute parent logic *)
SUPER^();

(* Run main state machine *)
StateMachine();

PROPERTY Active : REFERENCE TO BOOL
GET
Active REF= bActive;
END_GET
END_PROPERTY

PROPERTY ActiveCritical : REFERENCE TO UDINT
GET
ActiveCritical REF= iActiveCritical;
END_GET
END_PROPERTY

PROPERTY ActiveError : REFERENCE TO UDINT
GET
ActiveError REF= iActiveError;
END_GET
END_PROPERTY

PROPERTY ActiveInfo : REFERENCE TO UDINT
GET
ActiveInfo REF= iActiveInfo;
END_GET
END_PROPERTY

PROPERTY ActiveVerbose : REFERENCE TO UDINT
GET
ActiveVerbose REF= iActiveVerbose;
END_GET
END_PROPERTY

PROPERTY ActiveWarrning : REFERENCE TO UDINT
GET
ActiveWarrning REF= iActiveWarning;
END_GET
END_PROPERTY

PROPERTY AlarmsTable : REFERENCE TO ARRAY[1..iMAX_EVENTS] OF ST_Event
GET
AlarmsTable REF= arrActiveAlarms;
END_GET
END_PROPERTY

PROPERTY Busy : REFERENCE TO BOOL
GET
Busy REF= bBusy;
END_GET
END_PROPERTY

PROPERTY Error : REFERENCE TO BOOL
GET
Error REF= bError;
END_GET
END_PROPERTY

PROPERTY ErrorID : REFERENCE TO HRESULT
GET
ErrorID REF= iResult;
END_GET
END_PROPERTY

PROPERTY EventsTable : REFERENCE TO ARRAY[1..iMAX_EVENTS] OF ST_Event
GET
EventsTable REF= arrEvents;
END_GET
END_PROPERTY

PROPERTY FileName : STRING
GET
FileName := sFileName;
END_GET
SET
sFileName := FileName;
END_SET
END_PROPERTY

PROPERTY MaxEvents : UDINT
GET
MaxEvents := iMAX_EVENTS;
END_GET
END_PROPERTY

METHOD MR_Abort : BOOL
VAR_INPUT
END_VAR
IF eAlarmControlerState > ALARM_CONTROLER_UNINITIALIZED THEN
	bAbort := TRUE;
	MR_Abort := FALSE;
	bBusy := TRUE;
	
	eAlarmControlerState := ALARM_CONTROLER_ABORTING;
	fbMachineLogger.MR_AddLogs(CONCAT(sName,' : abort requested'));	
	
ELSIF eAlarmControlerState = ALARM_CONTROLER_UNINITIALIZED THEN
	bAbort := FALSE;
	MR_Abort := TRUE;
	bBusy := FALSE;
	bActive := FALSE;
	
	fbMachineLogger.MR_AddLogs(CONCAT(sName,' : abort done'));	
	
END_IF
END_METHOD

METHOD MR_Clear : BOOL
VAR_INPUT
	ipFilter : I_TcEventFilter;
	bResetConfirmation : BOOL;
END_VAR
IF eAlarmControlerState = ALARM_CONTROLER_IDLE THEN
	bClear := TRUE;
	MR_Clear := FALSE;
	bBusy := TRUE;
	THIS^.ipFilter := ipFilter;
	THIS^.bResetConfirmation := bResetConfirmation;
	
	eAlarmControlerState := ALARM_CONTROLER_CLEAR;
	fbMachineLogger.MR_AddLogs(CONCAT(sName,' : clear requested'));		
	
ELSIF eAlarmControlerState = ALARM_CONTROLER_CLEAR_DONE THEN
	bClear := FALSE;
	MR_Clear := TRUE;	
	bBusy := FALSE;
	
	fbMachineLogger.MR_AddLogs(CONCAT(sName,' : clear done'));		
	
END_IF
END_METHOD

METHOD MR_ClearAll : BOOL
VAR_INPUT
	bResetConfirmation : BOOL;
END_VAR
IF eAlarmControlerState = ALARM_CONTROLER_IDLE THEN
	bClearAll := TRUE;
	MR_ClearAll := FALSE;
	bBusy := TRUE;
	THIS^.bResetConfirmation := bResetConfirmation;
	
	eAlarmControlerState := ALARM_CONTROLER_CLEAR_ALL;
	fbMachineLogger.MR_AddLogs(CONCAT(sName,' : clear all requested'));		

ELSIF eAlarmControlerState = ALARM_CONTROLER_CLEAR_ALL_DONE THEN
	bClearAll := FALSE;
	MR_ClearAll := TRUE;
	bBusy := FALSE;
	
	fbMachineLogger.MR_AddLogs(CONCAT(sName,' : clear all done'));		
	
END_IF
END_METHOD

METHOD MR_Confirm : BOOL
VAR_INPUT
	ipFilter : I_TcEventFilter;
END_VAR
IF eAlarmControlerState = ALARM_CONTROLER_IDLE THEN
	bConfirm := TRUE;
	MR_Confirm := FALSE;
	bBusy := TRUE;
	THIS^.ipFilter := ipFilter;
	
	eAlarmControlerState := ALARM_CONTROLER_CONFIRM;
	fbMachineLogger.MR_AddLogs(CONCAT(sName,' : confirmation requested'));		
	
ELSIF eAlarmControlerState = ALARM_CONTROLER_CONFIRM_DONE THEN
	bConfirm := FALSE;
	MR_Confirm := TRUE;	
	bBusy := FALSE;
	
	fbMachineLogger.MR_AddLogs(CONCAT(sName,' : confirmation done'));		
	
END_IF
END_METHOD

METHOD MR_ConfirmAll : BOOL
VAR_INPUT
	bResetConfirmation : BOOL;
END_VAR
IF eAlarmControlerState = ALARM_CONTROLER_IDLE THEN
	bConfirmAll := TRUE;
	MR_ConfirmAll := FALSE;
	bBusy := TRUE;
	
	THIS^.bResetConfirmation := bResetConfirmation;
	eAlarmControlerState := ALARM_CONTROLER_CONFIRM_ALL;
	fbMachineLogger.MR_AddLogs(CONCAT(sName,' : confirmation of all requested'));		
	
ELSIF eAlarmControlerState = ALARM_CONTROLER_CONFIRM_ALL_DONE THEN
	bConfirmAll := FALSE;
	MR_ConfirmAll := TRUE;
	bBusy := FALSE;
	
	fbMachineLogger.MR_AddLogs(CONCAT(sName,' : confirmation of all done'));	
	
END_IF
END_METHOD

METHOD MR_Export : BOOL
VAR_INPUT
END_VAR
IF eAlarmControlerState = ALARM_CONTROLER_IDLE THEN
	bExport := TRUE;
	MR_Export := FALSE;
	bBusy := TRUE;
	
	eAlarmControlerState := ALARM_CONTROLER_EXPORT;
	fbMachineLogger.MR_AddLogs(CONCAT(sName,' : exportation requested'));	
	
ELSIF eAlarmControlerState = ALARM_CONTROLER_EXPORT_DONE THEN
	bExport := FALSE;
	MR_Export := TRUE;
	bBusy := FALSE;
	
	fbMachineLogger.MR_AddLogs(CONCAT(sName,' : exportation done'));	
	
END_IF
END_METHOD

METHOD MR_FirstCycle : BOOL
VAR_INPUT
	sName 		: STRING;
	sFileName 	: STRING;
END_VAR
THIS^.sName := sName;
THIS^.sFileName := sFileName;
END_METHOD

METHOD MR_Init : BOOL
VAR_INPUT
END_VAR
IF eAlarmControlerState = ALARM_CONTROLER_UNINITIALIZED THEN
	MR_Init := FALSE;
	bInit := TRUE;
	bBusy := TRUE;
	
	eAlarmControlerState := ALARM_CONTROLER_INITIALIZING;
	fbMachineLogger.MR_AddLogs(CONCAT(sName,' : initialization requested'));
	
ELSIF eAlarmControlerState = ALARM_CONTROLER_IDLE THEN
	bInit := FALSE;
	MR_Init := FALSE;
	bBusy := FALSE;
	bActive := TRUE;
	
	fbMachineLogger.MR_AddLogs(CONCAT(sName,' : initialization done'));
	
END_IF
END_METHOD

METHOD PROTECTED MS_Aborting
VAR_INPUT
END_VAR
Unsubscribe();
eAlarmControlerState := ALARM_CONTROLER_UNINITIALIZED;
END_METHOD

METHOD PROTECTED MS_Clear
VAR_INPUT
END_VAR
fbEventLogger.ConfirmAllAlarms(	nTimeStamp := 0);

iResult := fbEventLogger.ClearAlarms(	nTimeStamp 			:= 0,
										bResetConfirmation	:= bResetConfirmation,
										ipFilter 			:= ipFilter);

IF iResult = S_OK THEN
	eAlarmControlerState := ALARM_CONTROLER_CLEAR_DONE;
END_IF
END_METHOD

METHOD PROTECTED MS_ClearAll
VAR_INPUT
END_VAR
fbEventLogger.ConfirmAllAlarms(	nTimeStamp := 0);

iResult := fbEventLogger.ClearAllAlarms(	nTimeStamp := 0,
											bResetConfirmation := bResetConfirmation);

IF iResult = S_OK THEN
	eAlarmControlerState := ALARM_CONTROLER_CLEAR_ALL_DONE;
END_IF
END_METHOD

METHOD PROTECTED MS_ClearAllDone
VAR_INPUT
END_VAR
IF NOT bClearAll THEN
	eAlarmControlerState := ALARM_CONTROLER_IDLE;
END_IF
END_METHOD

METHOD PROTECTED MS_ClearDone
VAR_INPUT
END_VAR
IF NOT bClear THEN
	eAlarmControlerState := ALARM_CONTROLER_IDLE;
END_IF
END_METHOD

METHOD PROTECTED MS_Confirm
VAR_INPUT
END_VAR
iResult := fbEventLogger.ConfirmAlarms(	nTimeStamp	:= 0,
										ipFilter	:= ipFilter); 
										
IF iResult = S_OK THEN
	eAlarmControlerState := ALARM_CONTROLER_CONFIRM_DONE;
END_IF
END_METHOD

METHOD PROTECTED MS_ConfirmAll
VAR_INPUT
END_VAR
fbEventLogger.ConfirmAllAlarms(	nTimeStamp := 0);

iResult := fbEventLogger.ClearAllAlarms(	nTimeStamp := 0,
											bResetConfirmation := bResetConfirmation);
	
IF iResult = S_OK THEN
	eAlarmControlerState := ALARM_CONTROLER_CONFIRM_ALL_DONE;
END_IF
END_METHOD

METHOD PROTECTED MS_ConfirmAllDone
VAR_INPUT
END_VAR
IF NOT bConfirmAll THEN
	eAlarmControlerState := ALARM_CONTROLER_IDLE;
END_IF
END_METHOD

METHOD PROTECTED MS_ConfirmDone
VAR_INPUT
END_VAR
IF NOT bConfirm THEN
	eAlarmControlerState := ALARM_CONTROLER_IDLE;
END_IF
END_METHOD

METHOD PROTECTED MS_Export
VAR_INPUT
END_VAR
fbEventLogger.ExportLoggedEvents( 	sFileName := sFileName,
									ipExportSettings := 0,
									bError => bError,
									hrErrorCode => iResult);

IF iResult = S_OK THEN
	eAlarmControlerState := ALARM_CONTROLER_EXPORT_DONE;
END_IF
END_METHOD

METHOD PROTECTED MS_ExportDone
VAR_INPUT
END_VAR
IF NOT bExport THEN
	eAlarmControlerState := ALARM_CONTROLER_IDLE;
END_IF
END_METHOD

METHOD PROTECTED MS_Idle
VAR_INPUT
END_VAR
;
END_METHOD

METHOD PROTECTED MS_Initializing
VAR_INPUT
END_VAR
Subscribe(0, 0);
eAlarmControlerState := ALARM_CONTROLER_READY_INITIALIZED;
END_METHOD

METHOD PROTECTED MS_ReadyInitialized
VAR_INPUT
END_VAR
bActive := TRUE;
eAlarmControlerState := ALARM_CONTROLER_IDLE;
END_METHOD

METHOD PROTECTED MS_Uninitialized
VAR_INPUT
END_VAR
bActive := FALSE;
END_METHOD

PROPERTY Name : REFERENCE TO STRING
GET
Name REF= sName;
END_GET
END_PROPERTY

PROPERTY State : REFERENCE TO E_AlarmControlerState
GET
State REF= eAlarmControlerState;
END_GET
END_PROPERTY

METHOD PROTECTED StateMachine
VAR_INPUT
END_VAR
CASE eAlarmControlerState OF
	ALARM_CONTROLER_UNINITIALIZED:
		MS_Uninitialized();
	
	ALARM_CONTROLER_INITIALIZING:
		MS_Initializing();
		
	ALARM_CONTROLER_READY_INITIALIZED:
		MS_ReadyInitialized();	
	
	ALARM_CONTROLER_IDLE:
		MS_Idle();
		
	ALARM_CONTROLER_CONFIRM_ALL:
		MS_ConfirmAll();
		
	ALARM_CONTROLER_CONFIRM_ALL_DONE:
		MS_ConfirmAllDone();
	
	ALARM_CONTROLER_CLEAR_ALL:
		MS_ClearAll();
		
	ALARM_CONTROLER_CLEAR_ALL_DONE:
		MS_ClearAllDone();
		
	ALARM_CONTROLER_CONFIRM:
		MS_Confirm();
	
	ALARM_CONTROLER_CONFIRM_DONE:
		MS_ConfirmDone();
		
	ALARM_CONTROLER_CLEAR:
		MS_Clear();
		
	ALARM_CONTROLER_CLEAR_DONE:
		MS_ClearDone();
		
	ALARM_CONTROLER_EXPORT:
		MS_Export();
		
	ALARM_CONTROLER_EXPORT_DONE:
		MS_ExportDone();
		
	ALARM_CONTROLER_ABORTING:
		MS_Aborting();
		
END_CASE
END_METHOD

END_FUNCTION_BLOCK

// ---- POUs/Libs/Alarms/VisuEvents/FB_VisuEventsHandling.TcPOU
FUNCTION_BLOCK ABSTRACT FB_VisuEventsHandling EXTENDS FB_ListenerBase
VAR
	arrEvents				: ARRAY[1..iMAX_EVENTS] OF ST_Event;		//Dla HMI (* *)
	arrActiveAlarms			: ARRAY[1..iMAX_EVENTS] OF ST_Event;		//Dla HMI (*  *)
	arrActiveEvents			: ARRAY[1..iMAX_DEFINITION_EVENTS] OF ST_BaseEvent;	(*  *)
	
	iActiveDefinitionEvents	: UDINT;	(* zajetosc tabeli arrActiveEvents *)
	iActiveAlarms			: UDINT;	(* Zajetosc tabeli alarmow *)
	
	iActiveCritical			: UDINT;	(*  *)
	iActiveError			: UDINT;	(*  *)
	iActiveWarning			: UDINT;	(*  *)
	iActiveInfo				: UDINT;	(*  *)
	iActiveVerbose			: UDINT;	(*  *)
	
	bSummertime				: BOOL;		(*  *)
END_VAR

Execute();

METHOD Execute : HRESULT
VAR_INPUT
END_VAR
VAR_INST
	fbRequestEventText  : FB_RequestEventText;
	stBaseEvent 		: ST_BaseEvent;
	bReqText 			: BOOL;
	{attribute 'TcEncoding':='UTF-8'}
	sLastMessageText 	: STRING;
	index				: udint;
END_VAR
VAR
	rtAlarmCleard : R_TRIG;
END_VAR
Execute := SUPER^.Execute(); //retrieve events

IF iActiveDefinitionEvents > 0 AND bReqText = FALSE THEN
	stBaseEvent := arrActiveEvents[iActiveDefinitionEvents];
	fbRequestEventText.Request(eventClass:=stBaseEvent.guidEventClass, nEventId:=stBaseEvent.iEventId, nLangId := Tc3_EventLogger.GVL.nLangId_OnlineMonitoring, ipArgs:=stBaseEvent.iTcArguments);
	MEMSET(ADR(arrActiveEvents[iActiveDefinitionEvents]),0,SIZEOF(arrActiveEvents[iActiveDefinitionEvents]));
	iActiveDefinitionEvents := iActiveDefinitionEvents - 1;
	bReqText := TRUE;
END_IF

//retrieve the text of a message
IF 	bReqText AND fbRequestEventText.bError THEN 
	sLastMessageText := 'Error';
	bReqText := FALSE;
ELSIF bReqText AND NOT fbRequestEventText.bBusy THEN
	rtAlarmCleard(CLK := stBaseEvent.eEventType = E_EventType.ALARM_CLEARED); //RMA
	IF stBaseEvent.eEventType = E_EventType.MESSAGE OR stBaseEvent.eEventType = E_EventType.ALARM_RAISED THEN
		MEMCPY(ADR(arrEvents[2]),ADR(arrEvents[1]),SIZEOF(arrEvents[1]) * (iMAX_EVENTS - 1));
		fbRequestEventText.GetString(sLastMessageText, SIZEOF(sLastMessageText));
		arrEvents[1].iType := stBaseEvent.iType;
		arrEvents[1].eSeverity := stBaseEvent.eSeverity;
		arrEvents[1].iEventId := stBaseEvent.iEventId;
		arrEvents[1].guidEventClass := stBaseEvent.guidEventClass;
		arrEvents[1].sSourceName := stBaseEvent.sSourceName;
		arrEvents[1].iSourceID := stBaseEvent.iSourceID;
		//arrEvents[1].nTimeStamp := ULINT_TO_DT(stBaseEvent.nTimeStamp/10000000 - 11644473600); //100ns -> s - 1601.01.01:00:00:00
		arrEvents[1].iTimeStamp := stBaseEvent.iTimeStamp/10000 - 11644473600000; //100ns to ms -> /1000
		arrEvents[1].iTimeStampCleared := 0; //100ns to ms -> /1000
		arrEvents[1].iTimeStampConfirmed :=0; //100ns to ms -> /1000
		IF NOT bSummertime THEN
			arrEvents[1].iTimeStamp := arrEvents[1].iTimeStamp + 3600000;
		END_IF
		UTF8_TO_STRING(pDstSTRING:=ADR(arrEvents[1].sEventText), pSrcUTF8:=ADR(sLastMessageText), nDstSize:=SIZEOF(arrEvents[1].sEventText), nDstLen=> );
		IF LEN2(ADR(stBaseEvent.sJsonAttribute)) > 0 THEN
			//arrEvents[1].wsJsonAttribute := stBaseEvent.wsJsonAttribute;
			FindAndReplaceChar(
				pSrcString:= ADR(stBaseEvent.sJsonAttribute), 
				sDeleteChar:= '"', 
				sInsertChar:= '', 
				pDstString:= ADR(arrEvents[1].sJsonAttribute), 
				nDstSize:= LEN2(ADR(stBaseEvent.sJsonAttribute)));
			FindAndReplaceChar(
				pSrcString:= ADR(arrEvents[1].sJsonAttribute), 
				sDeleteChar:= ':', 
				sInsertChar:= '$T', 
				pDstString:= ADR(arrEvents[1].sJsonAttribute), 
				nDstSize:= LEN2(ADR(arrEvents[1].sJsonAttribute)));
			FindAndReplaceChar(
				pSrcString:= ADR(arrEvents[1].sJsonAttribute), 
				sDeleteChar:= ',', 
				sInsertChar:= '$N', 
				pDstString:= ADR(arrEvents[1].sJsonAttribute), 
				nDstSize:= LEN2(ADR(arrEvents[1].sJsonAttribute)));
			FindAndReplaceChar(
				pSrcString:= ADR(arrEvents[1].sJsonAttribute), 
				sDeleteChar:= '{', 
				sInsertChar:= '', 
				pDstString:= ADR(arrEvents[1].sJsonAttribute), 
				nDstSize:= LEN2(ADR(arrEvents[1].sJsonAttribute)));
			FindAndReplaceChar(
				pSrcString:= ADR(arrEvents[1].sJsonAttribute), 
				sDeleteChar:= '}', 
				sInsertChar:= '', 
				pDstString:= ADR(arrEvents[1].sJsonAttribute), 
				nDstSize:= LEN2(ADR(arrEvents[1].sJsonAttribute)));							
		END_IF	
		arrEvents[1].sEventText := arrEvents[1].sEventText;
		//aktywne alarmy
		IF stBaseEvent.eEventType = E_EventType.ALARM_RAISED THEN
			MEMCPY(ADR(arrActiveAlarms[2]),ADR(arrActiveAlarms[1]),SIZEOF(arrActiveAlarms[1]) * (iMAX_EVENTS - 1));
			arrActiveAlarms[1].iType 			:= arrEvents[1].iType;
			arrActiveAlarms[1].eSeverity 		:= arrEvents[1].eSeverity;
			arrActiveAlarms[1].iEventId 		:= arrEvents[1].iEventId;
			arrActiveAlarms[1].iTimeStamp 		:= arrEvents[1].iTimeStamp;
			arrActiveAlarms[1].sEventText 		:= arrEvents[1].sEventText;
			arrActiveAlarms[1].sJsonAttribute 	:= arrEvents[1].sJsonAttribute;
			arrActiveAlarms[1].guidEventClass 	:= arrEvents[1].guidEventClass;
			arrActiveAlarms[1].sSourceName 		:= arrEvents[1].sSourceName;
			arrActiveAlarms[1].iSourceID 		:= arrEvents[1].iSourceID;
			arrActiveAlarms[1].iTimeStampCleared := arrEvents[1].iTimeStampCleared;
			arrActiveAlarms[1].iTimeStampConfirmed := arrEvents[1].iTimeStampConfirmed;
			IF iActiveAlarms < iMAX_EVENTS THEN
				iActiveAlarms := iActiveAlarms + 1;
			END_IF
		END_IF
	ELSIF rtAlarmCleard.Q THEN
		//alarmy aktywne
		FOR index := 1 TO iActiveAlarms DO
			IF  GuidsEqualByVal(stBaseEvent.guidEventClass, arrActiveAlarms[index].guidEventClass) AND
				stBaseEvent.iEventId = arrActiveAlarms[index].iEventId AND 
				stBaseEvent.sSourceName = arrActiveAlarms[index].sSourceName AND 
				stBaseEvent.iSourceID = arrActiveAlarms[index].iSourceID THEN
				IF index < iMAX_EVENTS THEN
					MEMCPY(ADR(arrActiveAlarms[index]),ADR(arrActiveAlarms[index+1]),SIZEOF(arrActiveAlarms[1]) * (iActiveAlarms - index));
					MEMSET(ADR(arrActiveAlarms[iActiveAlarms]),0,SIZEOF(arrActiveAlarms[iActiveAlarms]));
					iActiveAlarms := iActiveAlarms - 1;
					EXIT;
				ELSE
					MEMSET(ADR(arrActiveAlarms[iActiveAlarms]),0,SIZEOF(arrActiveAlarms[iActiveAlarms]));
					iActiveAlarms := iActiveAlarms - 1;
				END_IF
			END_IF
		END_FOR
		//alarmy historyczne
		FOR index := 1 TO iMAX_EVENTS DO
			IF  GuidsEqualByVal(stBaseEvent.guidEventClass, arrEvents[index].guidEventClass) AND
				stBaseEvent.iEventId = arrEvents[index].iEventId AND 
				stBaseEvent.sSourceName = arrEvents[index].sSourceName AND 
				stBaseEvent.iSourceID = arrEvents[index].iSourceID THEN
				arrEvents[index].iTimeStampCleared := stBaseEvent.iTimeStamp/10000 - 11644473600000; //100ns to ms -> /1000
				IF NOT bSummertime THEN
					arrEvents[index].iTimeStampCleared := arrEvents[index].iTimeStampCleared + 3600000;
				END_IF
				EXIT;
			END_IF
		END_FOR
	ELSIF stBaseEvent.eEventType = E_EventType.ALARM_CONFIRMED THEN
		FOR index := 1 TO iMAX_EVENTS DO
			IF  GuidsEqualByVal(stBaseEvent.guidEventClass, arrActiveAlarms[index].guidEventClass) AND
				stBaseEvent.iEventId = arrActiveAlarms[index].iEventId AND 
				stBaseEvent.sSourceName = arrActiveAlarms[index].sSourceName AND 
				stBaseEvent.iSourceID = arrActiveAlarms[index].iSourceID THEN
				arrActiveAlarms[index].iTimeStampConfirmed := stBaseEvent.iTimeStamp/10000 - 11644473600000; //100ns to ms -> /1000
				IF NOT bSummertime THEN
					arrActiveAlarms[index].iTimeStampConfirmed := arrActiveAlarms[index].iTimeStampConfirmed + 3600000;
				END_IF
				EXIT;
			END_IF
		END_FOR	
		FOR index := 1 TO iMAX_EVENTS DO
			IF  GuidsEqualByVal(stBaseEvent.guidEventClass, arrEvents[index].guidEventClass) AND
				stBaseEvent.iEventId = arrEvents[index].iEventId AND 
				stBaseEvent.sSourceName = arrEvents[index].sSourceName AND 
				stBaseEvent.iSourceID = arrEvents[index].iSourceID THEN
				arrEvents[index].iTimeStampConfirmed := stBaseEvent.iTimeStamp/10000 - 11644473600000; //100ns to ms -> /1000
				IF NOT bSummertime THEN
					arrEvents[index].iTimeStampConfirmed := arrEvents[index].iTimeStampConfirmed + 3600000;
				END_IF
				EXIT;
			END_IF
		END_FOR	
	END_IF
	
	bReqText := FALSE;
END_IF
END_METHOD

METHOD OnAlarmCleared
VAR_INPUT
	fbEvent : REFERENCE TO FB_TcEvent;
END_VAR
IF iActiveDefinitionEvents >= iMAX_DEFINITION_EVENTS THEN
	RETURN; //skip new events
END_IF

MEMCPY(ADR(arrActiveEvents[2]),ADR(arrActiveEvents[1]),SIZEOF(arrActiveEvents[1]) * iActiveDefinitionEvents);
iActiveDefinitionEvents := iActiveDefinitionEvents + 1;
arrActiveEvents[1].iType := 1;
arrActiveEvents[1].guidEventClass := fbEvent.EventClass;
arrActiveEvents[1].eSeverity := fbEvent.eSeverity;
arrActiveEvents[1].iEventId := fbEvent.nEventId;
arrActiveEvents[1].iTimeStamp := fbEvent.nTimestamp;
arrActiveEvents[1].iTcArguments := fbEvent.ipArguments;
arrActiveEvents[1].eEventType := E_EventType.ALARM_CLEARED;
arrActiveEvents[1].sSourceName := fbEvent.ipSourceInfo.sName;
arrActiveEvents[1].iSourceID := fbEvent.ipSourceInfo.nId;
fbEvent.GetJsonAttribute(arrActiveEvents[1].sJsonAttribute, SIZEOF(arrActiveEvents[1].sJsonAttribute));

(* Active events type counter *)
IF arrActiveEvents[1].eSeverity = TcEventSeverity.Verbose THEN
	IF iActiveInfo > 0 THEN
		iActiveInfo := iActiveInfo - 1;	
	ELSE iActiveInfo :=0;
	END_IF
	
ELSIF arrActiveEvents[1].eSeverity = TcEventSeverity.Info THEN
	IF iActiveVerbose > 0 THEN
		iActiveVerbose := iActiveVerbose - 1;	
	ELSE iActiveVerbose := 0;
	END_IF
ELSIF arrActiveEvents[1].eSeverity = TcEventSeverity.Warning THEN
	IF iActiveWarning > 0 THEN
		iActiveWarning := iActiveWarning - 1;		
	ELSE iActiveWarning := 0;
	END_IF
	
ELSIF arrActiveEvents[1].eSeverity = TcEventSeverity.Error THEN
	IF iActiveError > 0 THEN
		iActiveError := iActiveError - 1;		
	ELSE iActiveError :=0;
	END_IF
	
ELSIF arrActiveEvents[1].eSeverity = TcEventSeverity.Critical THEN
	IF iActiveCritical > 0 THEN
		iActiveCritical := iActiveCritical - 1;	
	ELSE iActiveCritical := 0;
	END_IF
END_IF
END_METHOD

METHOD OnAlarmConfirmed
VAR_INPUT
	fbEvent : REFERENCE TO FB_TcEvent;
END_VAR
IF iActiveDefinitionEvents >= iMAX_DEFINITION_EVENTS THEN
	RETURN; //skip new events
END_IF

MEMCPY(ADR(arrActiveEvents[2]),ADR(arrActiveEvents[1]),SIZEOF(arrActiveEvents[1]) * iActiveDefinitionEvents);
iActiveDefinitionEvents := iActiveDefinitionEvents + 1;
arrActiveEvents[1].iType := 1;
arrActiveEvents[1].guidEventClass := fbEvent.EventClass;
arrActiveEvents[1].eSeverity := fbEvent.eSeverity;
arrActiveEvents[1].iEventId := fbEvent.nEventId;
arrActiveEvents[1].iTimeStamp := fbEvent.nTimestamp;
arrActiveEvents[1].iTcArguments := fbEvent.ipArguments;
arrActiveEvents[1].eEventType := E_EventType.ALARM_CONFIRMED;
arrActiveEvents[1].sSourceName := fbEvent.ipSourceInfo.sName;
arrActiveEvents[1].iSourceID := fbEvent.ipSourceInfo.nId;
fbEvent.GetJsonAttribute(arrActiveEvents[1].sJsonAttribute, SIZEOF(arrActiveEvents[1].sJsonAttribute));

(* Active events type counter *)
IF arrActiveEvents[1].eSeverity = TcEventSeverity.Verbose THEN
	IF iActiveInfo > 0 THEN
		iActiveInfo := iActiveInfo - 1;	
	ELSE 
		iActiveInfo :=0;
	END_IF
		
ELSIF arrActiveEvents[1].eSeverity = TcEventSeverity.Info THEN
	iActiveVerbose := iActiveVerbose - 1;	

ELSIF arrActiveEvents[1].eSeverity = TcEventSeverity.Warning THEN
	IF iActiveWarning > 0 THEN
		iActiveWarning := iActiveWarning - 1;
	ELSE iActiveWarning := 0;
	END_IF
			

ELSIF arrActiveEvents[1].eSeverity = TcEventSeverity.Error THEN
	IF iActiveError > 0 THEN
		iActiveError := iActiveError - 1;
	ELSE iActiveError := 0;	
	END_IF
	
ELSIF arrActiveEvents[1].eSeverity = TcEventSeverity.Critical THEN
	IF iActiveCritical > 0 THEN
		iActiveCritical := iActiveCritical - 1;	
	ELSE iActiveCritical := 0;
	END_IF
END_IF
END_METHOD

METHOD OnAlarmRaised
VAR_INPUT
	fbEvent : REFERENCE TO FB_TcEvent;
END_VAR
VAR
END_VAR
IF iActiveDefinitionEvents >= iMAX_DEFINITION_EVENTS THEN
	RETURN; //skip new events
END_IF

MEMCPY(ADR(arrActiveEvents[2]),ADR(arrActiveEvents[1]),SIZEOF(arrActiveEvents[1]) * iActiveDefinitionEvents);
iActiveDefinitionEvents := iActiveDefinitionEvents + 1;
arrActiveEvents[1].iType := 1;
arrActiveEvents[1].guidEventClass := fbEvent.EventClass;
arrActiveEvents[1].eSeverity := fbEvent.eSeverity;
arrActiveEvents[1].iEventId := fbEvent.nEventId;
arrActiveEvents[1].iTimeStamp := fbEvent.nTimestamp;
arrActiveEvents[1].iTcArguments := fbEvent.ipArguments;
arrActiveEvents[1].eEventType := E_EventType.ALARM_RAISED;
arrActiveEvents[1].sSourceName := fbEvent.ipSourceInfo.sName;
arrActiveEvents[1].iSourceID := fbEvent.ipSourceInfo.nId;
fbEvent.GetJsonAttribute(arrActiveEvents[1].sJsonAttribute, SIZEOF(arrActiveEvents[1].sJsonAttribute));

(* Active events type counter *)
IF arrActiveEvents[1].eSeverity = TcEventSeverity.Verbose THEN
	iActiveInfo := iActiveInfo + 1;	
	
ELSIF arrActiveEvents[1].eSeverity = TcEventSeverity.Info THEN
	IF iActiveVerbose < 4294967295 THEN
		iActiveVerbose := iActiveVerbose + 1;	
	ELSE iActiveVerbose := 4294967295;
	END_IF
	
ELSIF arrActiveEvents[1].eSeverity = TcEventSeverity.Warning THEN
	IF iActiveWarning < 4294967295 THEN
		iActiveWarning := iActiveWarning + 1;	
	ELSE iActiveWarning := 4294967295;
	END_IF
	
ELSIF arrActiveEvents[1].eSeverity = TcEventSeverity.Error THEN
	IF iActiveError < 4294967295 THEN
		iActiveError := iActiveError + 1;	
	ELSE iActiveError := 4294967295;
	END_IF
	
ELSIF arrActiveEvents[1].eSeverity = TcEventSeverity.Critical THEN
	IF iActiveCritical < 4294967295 THEN
		iActiveCritical := iActiveCritical + 1;	
	ELSE iActiveCritical := 4294967295;
	END_IF
	
END_IF
END_METHOD

METHOD OnMessageSent
VAR_INPUT
	fbEvent : REFERENCE TO FB_TcEvent;
END_VAR

VAR 
END_VAR
IF iActiveDefinitionEvents >= iMAX_DEFINITION_EVENTS THEN
	RETURN; //skip new events
END_IF

MEMCPY(ADR(arrActiveEvents[2]),ADR(arrActiveEvents[1]),SIZEOF(arrActiveEvents[1]) * iActiveDefinitionEvents);
iActiveDefinitionEvents := iActiveDefinitionEvents + 1;
arrActiveEvents[1].iType := 2;
arrActiveEvents[1].guidEventClass := fbEvent.EventClass;
arrActiveEvents[1].eSeverity := fbEvent.eSeverity;
arrActiveEvents[1].iEventId := fbEvent.nEventId;
arrActiveEvents[1].iTimeStamp := fbEvent.nTimestamp;
arrActiveEvents[1].iTcArguments := fbEvent.ipArguments;
arrActiveEvents[1].eEventType := E_EventType.MESSAGE;
arrActiveEvents[1].sSourceName := fbEvent.ipSourceInfo.sName;
arrActiveEvents[1].iSourceID := fbEvent.ipSourceInfo.nId;
fbEvent.GetJsonAttribute(arrActiveEvents[1].sJsonAttribute, SIZEOF(arrActiveEvents[1].sJsonAttribute));
END_METHOD

END_FUNCTION_BLOCK

// ---- POUs/Machine/Machine Control/PRG_MachineControl.TcPOU
PROGRAM PRG_MachineControl
VAR
	bFirstCycle 		: BOOL := TRUE;			(*  *)
	fbMachineControler 	: FB_MachineControl;	(*  *)
	fbFileLogger 		: FB_FileLogger;		(*	*)
END_VAR

IF bFirstCycle THEN
	bFirstCycle := FALSE;
	
	(* Assign machine controler reference to Shell API*)
	stShell.stPlatform.ref_fbMachineControler REF= fbMachineControler;
	
	(* Set assignamnet done bit for visu controler *)
	stShell.stFlags.bMachineCtrlAssignamentsDone := TRUE;
	
	fbMachineLogger.MR_FirstCycle( 	sName		:= 'PSE_Shell_Machine_Logger',
									sFileDir 	:= 'C:\TwinCAT\Tests\Loggers',
									sFileName 	:= 'PSE_Shell_Machine_Logger',
									sAmsNetId 	:= '',
									bAddTimeStamp := FALSE,
									bAddHeader := FALSE);
END_IF

IF NOT fbMachineLogger.Active THEN 
	fbMachineLogger.MR_Init();	
END_IF

(* Run global machine clock *)
fbMachineTime(bEnable := TRUE);
(* Cyclic run of machine controler *)
fbMachineControler();

fbMachineLogger();

END_PROGRAM

// ---- POUs/Machine/Machine Control/FB_MachineControl.TcPOU
FUNCTION_BLOCK FB_MachineControl EXTENDS FB_UniversalMachine IMPLEMENTS I_MachineControl
VAR
	iLoop : USINT;	(* for loop auxilary variable *)

	(* --- Sample actuators - from shell template --- DELETE IF NOT NEEDED - *)
	//arrDigitalInput		: ARRAY[0..19] OF FB_DigitalInput;			(* Array of sample digital inputs *)
	//arrDigitalOutput	: ARRAY[0..19] OF FB_DigitalOutput;			(* Array of sample digital outputs *)
	//arrCylinderDc		: ARRAY[0..9] OF FB_DoubleCoilCylinder;		(* Array of sample double coil cylinders *)
	//arrCylinderSc		: ARRAY[0..9] OF FB_SingleCoilCylinder;		(* Array of sample single coil cylinders *)
	//arrAxis				: ARRAY[0..19] OF FB_AxisServo;				(* Array of sample axis *)
	arrRobot			: FB_CR800EtherCAT;			(* Array of sample robots *)
	
	tonTestDelay	: TON;	(* Delay which allows to see any page changes during tests *)
	
	(* --- Sample actuators - from shell template --- DELETE IF NOT NEEDED - *)	
	bStart			: BOOL;
	
	(* CR800 - testing *)
	lrPositionX1 : LREAL := 203.733;
	lrPositionY1 : LREAL := 100.000;
	lrRotation1  : LREAL := 216.699;
	
	lrPositionX2 : LREAL := -13.733;
	lrPositionY2 : LREAL := 8.001;
	lrRotation2  : LREAL := -2.889;
	
	
	bUserDefinedArea1	: BOOL;
	bTryIt1				: BOOL;
	bTryIt2				: BOOL;
	
	(* State machines *)
	
	eMachineStateUninitialized						: E_MachineCtrlStateUninitialized;
	
	(* CR800 EtherCAT diagnostic *) 	                                                                
	fbGetCR800EcState				:  FB_EcGetSlaveState;		
	fbSetCR800CtrlState 			:  FB_EcReqSlaveState;		
	stCR800GetEcState				:  ST_EcSlaveState;		
	(* Robots EtherCAT communication *)                      		
	sPLC_NET_ID 							: STRING:= '192.168.152.1.3.1';//'5.87.101.228.3.1'; hardware config							
	iCR800_1_ADDRESS						: UINT	:= 1015; //hardware config										
	iCR800_2_ADDRESS						: UINT	:= 1016; //hardware config
END_VAR

IF bFirstCycle THEN
	(* bFirstCycle bit reset by parent *)
	(* --- Assign initial parameters for machine objects ---*)
	(* ---- DELETE IF NOT NEEDED ---- *)
	(* Assign sample digital inputs *)
//	FOR iLoop := 0 TO 19 DO
//		arrDigitalInput[iLoop].MR_FirstCycle(CONCAT('Digital_Input_',USINT_TO_STRING(iLoop)),CONCAT('EL1008-',USINT_TO_STRING(iLoop/8)),USINT_TO_STRING(iLoop MOD 8));
//	END_FOR
	
//	(* Assign sample digital outputs *)
//	FOR iLoop := 0 TO 19 DO
//		arrDigitalOutput[iLoop].MR_FirstCycle(CONCAT('Digital_Output_',USINT_TO_STRING(iLoop)),CONCAT('EL2008-',USINT_TO_STRING(iLoop/8)),USINT_TO_STRING(iLoop MOD 8));
//	END_FOR
	
//	(* Assign sample cylinders *)
//	FOR iLoop := 0 TO 9 DO
//		arrCylinderDc[iLoop].MR_FirstCycle(	sName					:= CONCAT('Double_Coil_Cylinder_',USINT_TO_STRING(iLoop)),
//											sActiveSensorModuleType :=CONCAT('EL1008-',USINT_TO_STRING(iLoop/4)),
//											sActiveSensorPortID 	:= USINT_TO_STRING(iLoop*2),
//											sHomeSensorModuleType	:=CONCAT('EL1008-',USINT_TO_STRING(iLoop/4)),
//											sHomeSensorPortID		:= USINT_TO_STRING(iLoop*2+1),
//											tGoHomeTimeout			:= T#10S,
//											tGoActiveTimeout		:= T#10S,
//											tDelay 					:= T#1S);
//		arrCylinderDc[iLoop].Simulation := TRUE;
//		arrCylinderDc[iLoop].ref_poActiveValve.ModuleType := CONCAT('EL2008-',USINT_TO_STRING(iLoop/4));
//		arrCylinderDc[iLoop].ref_poActiveValve.PortID := USINT_TO_STRING(iLoop*2);
//		arrCylinderDc[iLoop].ref_poHomeValve.ModuleType := CONCAT('EL2008-',USINT_TO_STRING(iLoop/4));
//		arrCylinderDc[iLoop].ref_poHomeValve.PortID := USINT_TO_STRING(iLoop*2+1);
//	END_FOR
	
//	FOR iLoop := 0 TO 9 DO
//		arrCylinderSc[iLoop].MR_FirstCycle(	sName				:= CONCAT('Single_Coil_Cylinder_', USINT_TO_STRING(iLoop)),
//											sActiveSensorModuleType :=CONCAT('EL1008-',USINT_TO_STRING(iLoop/4)),
//											sActiveSensorPortID :=USINT_TO_STRING(iLoop*2),
//											sHomeSensorModuleType :=CONCAT('EL1008-',USINT_TO_STRING(iLoop/4)),
//											sHomeSensorPortID	:=USINT_TO_STRING(iLoop*2+1),
//											tGoHomeTimeout 		:= T#12S,
//											tGoActiveTimeout 	:= T#12S,
//											tDelay 				:= T#2S);
//		arrCylinderSc[iLoop].Simulation := TRUE;
//		arrCylinderSc[iLoop].ref_poActiveValve.ModuleType := CONCAT('EL2008-',USINT_TO_STRING(iLoop/8));
//		arrCylinderSc[iLoop].ref_poActiveValve.PortID := USINT_TO_STRING(iLoop);
//	END_FOR
	
//	(* Assign sample axes *)
//	FOR iLoop := 0 TO 19 DO
//		arrAxis[iLoop].MR_FirstCycle( 	sName 				:= CONCAT('Axis_',USINT_TO_STRING(iLoop)),
//										sMeasurementUnits 	:= 'mm',
//										bModulo				:= FALSE);
//		arrAxis[iLoop].ref_HomeSwitch.ModuleType :=CONCAT('EL1008-',USINT_TO_STRING(iLoop/8));
//		arrAxis[iLoop].ref_HomeSwitch.PortID :=USINT_TO_STRING(iLoop MOD 8);			
//	END_FOR	
	
	(* Assign sample robots *)
	//FOR iLoop := 0 TO 0 DO
		arrRobot.MR_FirstCycle(	sName		:= 'Robot 1',
								iOverride	:= 5);
	//END_FOR
	(* ---- DELETE IF NOT NEEDED ---- *)
END_IF

(* Execute parent implementation *)
SUPER^();

(* --- Cyclic run of internal objects ---*)
(* ---- DELETE IF NOT NEEDED ---- *)
//(* Cyclic run of sample inputs *)
//FOR iLoop := 0 TO 19 DO
//	arrDigitalInput[iLoop]();
//END_FOR

//(* Cyclic run of sample outputs *)
//FOR iLoop := 0 TO 19 DO
//	arrDigitalOutput[iLoop]();
//END_FOR
	
//(* Cyclic run of sample double coil cylinders *)
//FOR iLoop := 0 TO 9 DO
//	arrCylinderDc[iLoop]();
//END_FOR

//(* Cyclic run of sample single coil cylinders *)
//FOR iLoop := 0 TO 9 DO
//	arrCylinderSc[iLoop]();
//END_FOR

//(* Cyclic run of sample axis *)
//FOR iLoop := 0 TO 19 DO
//	arrAxis[iLoop]();
//END_FOR

(* Cyclic run of sample robots *)
//FOR iLoop := 0 TO 9 DO
	arrRobot();
//END_FOR

IF bTryIt1 THEN
	arrRobot.MR_SendPosition1( lrPositionX1 := lrPositionX1,
								lrPositionY1 := lrPositionY1,
								lrRotation1  := lrRotation1);
	IF NOT arrRobot.SendingPosition1 THEN
		bTryIt1 := FALSE;
	END_IF
END_IF

IF bTryIt2 THEN
	arrRobot.MR_SendPosition2( lrPositionX2 := lrPositionX2,
								lrPositionY2 := lrPositionY2,
								lrRotation2  := lrRotation2);
	IF NOT arrRobot.SendingPosition2 THEN
		bTryIt1 := FALSE;
	END_IF
END_IF

bUserDefinedArea1 := arrRobot.UserDefinedArea1;

tonTestDelay();
(* ---- DELETE IF NOT NEEDED ---- *)

METHOD MR_Start : BOOL
VAR_INPUT
END_VAR
bRunning := TRUE;

IF NOT bStart THEN
	fbMsgAutoStarted.Send(0);
	bStart := TRUE;
END_IF
END_METHOD

METHOD MR_Stop : BOOL
VAR_INPUT
END_VAR
bRunning := FALSE;

IF bStart THEN
	fbMsgAutoStopped.Send(0);
	bStart := FALSE;
END_IF
END_METHOD

METHOD PROTECTED MS_Aborting
VAR_INPUT
END_VAR
(* 
Add here code to abort all machine objects's e.g robots, axes, cylinders. 
At the end add "eMachineState := MACHINE_STATE_UNINITIALIZED;" to finish aborting.
*)
(* Aborting simulation - DELETE *)
tonTestDelay(IN := TRUE, PT:= T#4S);
IF tonTestDelay.Q THEN
	tonTestDelay(IN := FALSE);
	eMachineState := MACHINE_STATE_UNINITIALIZED;
END_IF
END_METHOD

METHOD PROTECTED MS_Auto
VAR_INPUT
END_VAR
(* 
Add here code to perform automatic process.
*)
;
END_METHOD

METHOD PROTECTED MS_AutoToManual
VAR_INPUT
END_VAR
(* 
Add here code to switch machine into manual mode. 
At the end add "eMachineState := MACHINE_STATE_MANUAL;" to finish switching.
*)
(* Switching mode to manual simulation - DELETE *)
tonTestDelay(IN := TRUE, PT:= T#4S);
bRunning := FALSE;
IF tonTestDelay.Q THEN
	tonTestDelay(IN := FALSE);
	eMachineState := MACHINE_STATE_MANUAL;
END_IF
END_METHOD

METHOD PROTECTED MS_Emergency
VAR_INPUT
END_VAR
END_METHOD

METHOD PROTECTED MS_Initializing
VAR_INPUT
END_VAR
(* 
Add here code to initialize all machine objects's e.g robots, axes, cylinders. 
At the end add "eMachineState := MACHINE_STATE_READY_INITIALIZED;" to finish initialization.
*)
(* Initialization simulation - DELETE  *)
tonTestDelay(IN := TRUE, PT:= T#4S);
IF tonTestDelay.Q THEN
	tonTestDelay(IN := FALSE);
	eMachineState := MACHINE_STATE_READY_INITIALIZED;
END_IF
END_METHOD

METHOD PROTECTED MS_Manual
VAR_INPUT
END_VAR
(* 
Leave empty - manual mode is provided by HMI controler and automatic frame generator.
*)
;
END_METHOD

METHOD PROTECTED MS_ManualToAuto
VAR_INPUT
END_VAR
(* 
Add here code to switch machine into auto mode. 
At the end add "eMachineState := MACHINE_STATE_MANUAL;" to finish switching.
*)
(* Switching mode to auto simulation - DELETE *)
tonTestDelay(IN := TRUE, PT:= T#4S);
IF tonTestDelay.Q THEN
	tonTestDelay(IN := FALSE);
	eMachineState := MACHINE_STATE_AUTO;
END_IF
END_METHOD

METHOD PROTECTED MS_ReadyInitialized
VAR_INPUT
END_VAR
(*
Add code here if some internal parameters are needed to set after initialization or leave it default.
At the end add "eMachineState := MACHINE_STATE_AUTO;" to finish and go to IDLE state.
*)
(* Ready-Initialized simulation - DELETE  *)
tonTestDelay(IN := TRUE, PT:= T#4S);
IF tonTestDelay.Q THEN
	tonTestDelay(IN := FALSE);
	eMachineState := MACHINE_STATE_AUTO;
END_IF
END_METHOD

METHOD PROTECTED MS_Reset
VAR_INPUT
END_VAR
(* 
Add here code to reset all machine objects's e.g robots, axes, cylinders. 
At the end add "eMachineState := MACHINE_STATE_RESET_DONE;" to finish reseting.
*)
(* Reset simulation - DELETE  *)
tonTestDelay(IN := TRUE, PT:= T#4S);
IF tonTestDelay.Q THEN
	tonTestDelay(IN := FALSE);
	eMachineState := MACHINE_STATE_RESET_DONE;
END_IF
END_METHOD

METHOD PROTECTED MS_ResetDone
VAR_INPUT
END_VAR
eMachineState := eMachineStateBeforeReset;
END_METHOD

METHOD PROTECTED MS_Uninitialized
VAR_INPUT
END_VAR
CASE eMachineStateUninitialized OF
	MACHINE_STATE_UNINITIALIZED_CR800_ETHERCAT_STATUS_CHECK:
		fbGetCR800EcState(			sNetId 		:= sPLC_NET_ID,
									nSlaveAddr	:= iCR800_1_ADDRESS,
									bExecute	:= TRUE,
									tTimeout 	:= DEFAULT_ADS_TIMEOUT,
									state		=> stCR800GetEcState);
		IF NOT fbGetCR800EcState.bBusy AND NOT fbGetCR800EcState.bError THEN
			fbGetCR800EcState(bExecute := FALSE);
			eMachineStateUninitialized := MACHINE_STATE_UNINITIALIZED_CR800_ETHERCAT_STATUS_CHECK_DONE;
		END_IF
	
	MACHINE_STATE_UNINITIALIZED_CR800_ETHERCAT_STATUS_CHECK_DONE:
		IF stCR800GetEcState.deviceState = EC_DEVICE_STATE_ERROR OR stCR800GetEcState.deviceState = 84 THEN
			eMachineStateUninitialized := MACHINE_STATE_UNINITIALIZED_CR800_ETHERCAT_ERROR_RESET;
			
		ELSIF stCR800GetEcState.deviceState = EC_DEVICE_STATE_SAFEOP THEN
			eMachineStateUninitialized := MACHINE_STATE_UNINITIALIZED_CR800_ETHERCAT_REQUEST_OP_STATE;
			
		ELSIF stCR800GetEcState.deviceState = EC_DEVICE_STATE_OP THEN
			eMachineStateUninitialized := MACHINE_STATE_UNINITIALIZED_CR800_CHECK_POWER_REGISTER;		
		ELSE
			eMachineStateUninitialized := MACHINE_STATE_UNINITIALIZED_CR800_ETHERCAT_STATUS_CHECK;
		END_IF
		
	MACHINE_STATE_UNINITIALIZED_CR800_ETHERCAT_ERROR_RESET:
		fbSetCR800CtrlState( 		sNetId 		:= sPLC_NET_ID,
									nSlaveAddr	:= iCR800_1_ADDRESS,
									bExecute 	:= TRUE,
									tTimeout 	:= DEFAULT_ADS_TIMEOUT,
									state 		:= EC_DEVICE_STATE_ERROR);
		IF NOT fbSetCR800CtrlState.bBusy AND NOT fbSetCR800CtrlState.bError THEN
			fbSetCR800CtrlState(bExecute := FALSE);
			eMachineStateUninitialized := MACHINE_STATE_UNINITIALIZED_CR800_ETHERCAT_STATUS_CHECK;
		END_IF
		
	MACHINE_STATE_UNINITIALIZED_CR800_ETHERCAT_REQUEST_OP_STATE:
		fbSetCR800CtrlState( 		sNetId 		:= sPLC_NET_ID,
									nSlaveAddr	:= iCR800_1_ADDRESS,
									bExecute 	:= TRUE,
									tTimeout 	:= DEFAULT_ADS_TIMEOUT,
									state 		:= EC_DEVICE_STATE_OP);
		IF NOT fbSetCR800CtrlState.bBusy AND NOT fbSetCR800CtrlState.bError THEN
			fbSetCR800CtrlState(bExecute := FALSE);
			eMachineStateUninitialized := MACHINE_STATE_UNINITIALIZED_CR800_ETHERCAT_STATUS_CHECK;
		END_IF
		
	MACHINE_STATE_UNINITIALIZED_CR800_CHECK_POWER_REGISTER:
		IF arrRobot.CR800PoweredOn THEN
			eMachineStateUninitialized := MACHINE_STATE_UNINITIALIZED_DONE;
		END_IF
		
	MACHINE_STATE_UNINITIALIZED_DONE:
		;
END_CASE
END_METHOD

PROPERTY Robots : REFERENCE TO FB_CR800EtherCAT
GET
Robots REF= arrRobot;
END_GET
END_PROPERTY

END_FUNCTION_BLOCK

// ---- POUs/Libs/Platform/Universal Machine/FB_UniversalMachine.TcPOU
(* 
:Description: This function block is base for of machine control module in all projects.
*)
FUNCTION_BLOCK ABSTRACT FB_UniversalMachine IMPLEMENTS I_UniversalMachine
VAR
	bFirstCycle		: BOOL := TRUE;							(*  *)
	bInit			: BOOL;									(*  *)
	bAbort 			: BOOL;									(*  *)
	bReset 			: BOOL;									(*  *)
	bSwitchToAuto 	: BOOL;									(*  *)
	bSwitchToManual : BOOL;									(*  *)
	bStepMode		: BOOL;									(*  *)
	
	bActive			: BOOL;									(*  *)
	bRunning		: BOOL;
	bError			: BOOL;									(*  *)
	iErrorID		: UDINT;								(*  *)

	eMachineState 				: E_MachineCtrlState;		(*  *)
	eMachineStateBeforeReset	: E_MachineCtrlState;		(*  *)
	
	(* Tc3 EventLogger - messages *)
	fbMsgInitStarted 			: FB_TcMessage;				(*  *)
	fbMsgInitDone 				: FB_TcMessage;				(*  *)
	fbMsgInAutoMode				: FB_TcMessage;				(*  *)
	fbMsgSwitchingToManual		: FB_TcMessage;				(*  *)
	fbMsgInManualMode			: FB_TcMessage;				(*  *)
	fbMsgSwitcingToAuto			: FB_TcMessage;				(*  *)
	fbMsgAutoStarted			: FB_TcMessage;				(*  *)
	fbMsgAutoStopped			: FB_TcMessage;				(*  *)
	fbMsgReset					: FB_TcMessage;				(*  *)
	fbMsgResetDone				: FB_TcMessage;				(*  *)
	fbMsgAbort					: FB_TcMessage;				(*  *)
	fbMsgAbortDone				: FB_TcMessage;				(*  *)
	
	fbSource					: FB_TcSourceInfo;
	
	hr							: HRESULT;
	
	rtError		: R_TRIG; 					(* Rising edge trigger for function block error *)
END_VAR
(*
Version history:

+-------------+------------+----------------+----------+------------------------------------------+
|Date         | Version    | created under  | Author   | Remark                                   |
+=============+============+================+==========+==========================================+
|2022-02      | 1.0.0.0    | V3.1.4024.22   | ADBO     | Function block created                   |
+-------------+------------+----------------+----------+------------------------------------------+

*)

IF bFirstCycle THEN
	bFirstCycle := FALSE;
	
	fbMsgInitStarted.CreateEx( stEventEntry := TC_EVENTS.ShellMachineEventClass.InitStarted, ipSourceInfo := 0);
								
	fbMsgInitDone.CreateEx( stEventEntry := TC_EVENTS.ShellMachineEventClass.InitDone, ipSourceInfo := 0);
								
	fbMsgInAutoMode.CreateEx( stEventEntry := TC_EVENTS.ShellMachineEventClass.InAutoMode, ipSourceInfo := 0);
								
	fbMsgSwitchingToManual.CreateEx( stEventEntry := TC_EVENTS.ShellMachineEventClass.SwitchingToManual, ipSourceInfo := 0);
								
	fbMsgInManualMode.CreateEx( stEventEntry := TC_EVENTS.ShellMachineEventClass.InManualMode, ipSourceInfo := 0);
								
	fbMsgAutoStarted.CreateEx( stEventEntry := TC_EVENTS.ShellMachineEventClass.AutoStarted, ipSourceInfo := 0);
								
	fbMsgAutoStopped.CreateEx( stEventEntry := TC_EVENTS.ShellMachineEventClass.AutoStopped, ipSourceInfo := 0);
								
	fbMsgReset.CreateEx( stEventEntry := TC_EVENTS.ShellMachineEventClass.Reset, ipSourceInfo := 0);
								
	fbMsgResetDone.CreateEx( stEventEntry := TC_EVENTS.ShellMachineEventClass.ResetDone, ipSourceInfo := 0);
								
	fbMsgAbort.CreateEx( stEventEntry := TC_EVENTS.ShellMachineEventClass.Abort, ipSourceInfo := 0);
								
	fbMsgAbortDone.CreateEx( stEventEntry := TC_EVENTS.ShellMachineEventClass.AbortDone, ipSourceInfo := 0);
	
END_IF

(* Set status flags *)
bActive := eMachineState >= MACHINE_STATE_AUTO;

(* Report errors that occur *)
rtError(CLK:=bError);

IF rtError.Q THEN 
	fbMachineLogger.MR_AddLogs(FUN_MergeStrings5('Universal_Machine', ' : Error occured (error ID: ', UDINT_TO_STRING(iErrorID), ')', ''));
END_IF

(* Run standard state machine *)
StateMachine();

PROPERTY Active : REFERENCE TO BOOL
GET
Active REF= bActive;
END_GET
END_PROPERTY

PROPERTY Error : REFERENCE TO BOOL
GET
Error REF= bError;
END_GET
END_PROPERTY

METHOD MR_Abort : BOOL
VAR_INPUT
END_VAR
IF eMachineState > MACHINE_STATE_UNINITIALIZED THEN
	bAbort := FALSE;
	MR_Abort := FALSE;
	fbMsgAbort.Send(0);
	fbMachineLogger.MR_AddLogs(CONCAT('Main machine controller',' : abort requested'));	
	eMachineState := MACHINE_STATE_ABORTING;
	
ELSIF eMachineState = MACHINE_STATE_UNINITIALIZED THEN
	bAbort := TRUE;
	MR_Abort := TRUE;
	fbMsgAbortDone.Send(0);	
	fbMachineLogger.MR_AddLogs(CONCAT('Main machine controller',' : abort done'));	
	
END_IF
END_METHOD

METHOD MR_Init : BOOL
VAR_INPUT
END_VAR
IF eMachineState = MACHINE_STATE_UNINITIALIZED THEN
	bInit := TRUE;
	MR_Init := FALSE;
	fbMsgInitStarted.Send(0);
	fbMachineLogger.MR_AddLogs(CONCAT('Main machine controller',' : initialization requested'));	
	eMachineState := MACHINE_STATE_INITIALIZING;
	
ELSIF eMachineState = MACHINE_STATE_AUTO AND bInit THEN
	bInit := FALSE;
	MR_Init := TRUE;
	fbMsgInitDone.Send(0);
	fbMachineLogger.MR_AddLogs(CONCAT('Main machine controller',' : initialization done'));	

END_IF
END_METHOD

METHOD MR_Reset : BOOL
VAR_INPUT
END_VAR
IF eMachineState = MACHINE_STATE_AUTO THEN
	bReset := TRUE;
	MR_Reset := FALSE;
	fbMsgReset.Send(0);
	fbMachineLogger.MR_AddLogs(CONCAT('Main machine controller',' : reset requested'));
	eMachineState := MACHINE_STATE_RESET;
	
ELSIF eMachineState = MACHINE_STATE_RESET_DONE THEN
	bReset := FALSE;
	MR_Reset := TRUE;
	fbMsgResetDone.Send(0);
	fbMachineLogger.MR_AddLogs(CONCAT('Main machine controller',' : reset done'));

END_IF
END_METHOD

METHOD ABSTRACT MR_Start : BOOL
VAR_INPUT
END_VAR
END_METHOD

METHOD ABSTRACT MR_Stop : BOOL
VAR_INPUT
END_VAR
END_METHOD

METHOD MR_SwitchToAuto : BOOL
VAR_INPUT
END_VAR
IF eMachineState = MACHINE_STATE_MANUAL THEN
	bSwitchToAuto := TRUE;
	MR_SwitchToAuto := FALSE;
	fbMsgSwitcingToAuto.Send(0);
	fbMachineLogger.MR_AddLogs(CONCAT('Main machine controller',' : switching to auto requested'));
	eMachineState := MACHINE_STATE_MANUAL_TO_AUTO;
	
ELSIF eMachineState = MACHINE_STATE_AUTO THEN
	bSwitchToAuto := FALSE;
	MR_SwitchToAuto := TRUE;
	fbMsgInAutoMode.Send(0);
	fbMachineLogger.MR_AddLogs(CONCAT('Main machine controller',' : switching to auto done'));

END_IF
END_METHOD

METHOD MR_SwitchToManual : BOOL
VAR_INPUT
END_VAR
IF eMachineState = MACHINE_STATE_AUTO THEN
	bSwitchToManual := TRUE;
	MR_SwitchToManual := FALSE;
	fbMsgSwitchingToManual.Send(0);
	fbMachineLogger.MR_AddLogs(CONCAT('Main machine controller',' : switching to manual requested'));
	eMachineState := MACHINE_STATE_AUTO_TO_MANUAL;
	
ELSIF eMachineState = MACHINE_STATE_MANUAL THEN
	bSwitchToManual := FALSE;
	MR_SwitchToManual := TRUE;
	fbMsgInManualMode.Send(0);
	fbMachineLogger.MR_AddLogs(CONCAT('Main machine controller',' : switching to manual done'));

END_IF
END_METHOD

METHOD PROTECTED ABSTRACT MS_Aborting
VAR_INPUT
END_VAR
END_METHOD

METHOD PROTECTED ABSTRACT MS_Auto
VAR_INPUT
END_VAR
END_METHOD

METHOD PROTECTED ABSTRACT MS_AutoToManual
VAR_INPUT
END_VAR
END_METHOD

METHOD PROTECTED ABSTRACT MS_Emergency
VAR_INPUT
END_VAR
END_METHOD

METHOD PROTECTED ABSTRACT MS_Initializing
VAR_INPUT
END_VAR
END_METHOD

METHOD PROTECTED ABSTRACT MS_Manual
VAR_INPUT
END_VAR
END_METHOD

METHOD PROTECTED ABSTRACT MS_ManualToAuto
VAR_INPUT
END_VAR
END_METHOD

METHOD PROTECTED ABSTRACT MS_ReadyInitialized
VAR_INPUT
END_VAR
END_METHOD

METHOD PROTECTED ABSTRACT MS_Reset
VAR_INPUT
END_VAR
END_METHOD

METHOD PROTECTED ABSTRACT MS_ResetDone
VAR_INPUT
END_VAR
END_METHOD

METHOD PROTECTED ABSTRACT MS_Uninitialized
VAR_INPUT
END_VAR
END_METHOD

PROPERTY Running : REFERENCE TO BOOL
GET
Running REF= bRunning;
END_GET
END_PROPERTY

PROPERTY State : REFERENCE TO E_MachineCtrlState
GET
State REF= eMachineState;
END_GET
END_PROPERTY

METHOD PROTECTED StateMachine
VAR_INPUT
END_VAR
CASE eMachineState OF
	(* Machine is not ready to work *)
	MACHINE_STATE_UNINITIALIZED:
		MS_Uninitialized();
		
	(* Initialization in progress *)
	MACHINE_STATE_INITIALIZING:
		MS_Initializing();
		
	(* Initialization finished *)
	MACHINE_STATE_READY_INITIALIZED:
		MS_ReadyInitialized();
	
	(* Machine in automatic mode *)
	MACHINE_STATE_AUTO:
		MS_Auto();
	
	(* Safe switch from automatic to manual mode*)
	MACHINE_STATE_AUTO_TO_MANUAL:
		MS_AutoToManual();
	
	(* Machie in manual mode *)
	MACHINE_STATE_MANUAL:
		MS_Manual();
	
	(* Safe switch from manual to automatic mode *)
	MACHINE_STATE_MANUAL_TO_AUTO:
		MS_ManualToAuto();
		
	(* Safe switch from manual to automatic mode *)
	MACHINE_STATE_RESET:
		MS_Reset();
		
	(* Safe switch from manual to automatic mode *)
	MACHINE_STATE_RESET_DONE:
		MS_ResetDone();
		
	(* Safe deintialization of machine *)
	MACHINE_STATE_ABORTING:
		MS_Aborting();
		
	(* Machine safety mode *)
	MACHINE_STATE_EMERGENCY:
		MS_Emergency();
		
END_CASE
END_METHOD

END_FUNCTION_BLOCK

// ---- POUs/Libs/Utilities/StringMerge/FUN_MergeStrings5.TcPOU
(* 
:Description: This function is used to merge 5 strings
*)
FUNCTION FUN_MergeStrings5 : STRING
VAR_INPUT
	sStr1	: STRING;		(* First string in merge row *)
	sStr2	: STRING;		(* Second string in merge row *)
	sStr3	: STRING;		(* Third string in merge row *)
	sStr4	: STRING;		(* Fourth string in merge row *)
	sStr5	: STRING;		(* Fifth string in merge row *)

END_VAR

FUN_MergeStrings5 := CONCAT(sStr1,sStr2);
FUN_MergeStrings5 := CONCAT(FUN_MergeStrings5, sStr3);
FUN_MergeStrings5 := CONCAT(FUN_MergeStrings5, sStr4);
FUN_MergeStrings5 := CONCAT(FUN_MergeStrings5, sStr5);

END_FUNCTION

// ---- POUs/Libs/Robots/Mitsubishi/FB_CR800EtherCAT.TcPOU
FUNCTION_BLOCK FB_CR800EtherCAT IMPLEMENTS I_CR800EtherCAT
VAR CONSTANT
	iMIN_ETHERCAT_REGISTER_IN_CR800	: INT 	:= 6000 ;	(*  *)
	iMAX_ETHERCAT_REGISTER_IN_CR800	: INT 	:= 6255 ;	(*  *)
	
	iSEND_REQUEST_ADDRESS			: UINT 	:= 6030 ;	(*  *)
	iRECEIVE_REQUEST_ADDRESS		: UINT 	:= 6031 ;	(*  *)
	
	tWATCHDOG_TIMEOUT				: TIME 	:= T#2S ;	(* Input timeout *)
END_VAR
VAR
	bFirstCycle			: BOOL := TRUE;	(* First cycle procedure bit *)
	sName				: STRING;		(*  *)
	
	stCR800EthercatData : ST_CR800EthercatData ;(* Data to map *)
	
	(* Internal commands *)
	bIsHomed					: BOOL;			(* Robot is it's home postion *)
	bReset						: BOOL;			(* Reset function block *)
	
	(* CR800 state *)
	bInit 						: BOOL;			(* Prepare a CR800 to work *)
	bGoHome 					: BOOL;			(* Moves a robot to the home postion *)
	bUpdateRecipes				: BOOL;			(* CR800 is updating recpies*)
	bGoAuto						: BOOL;			(* Robot goes to auto mode*)
	bDoAction					: BOOL;			(* Robot is doing action in automode*)
	bCycleStop					: BOOL;			(* Cr800 cycle is stopping *)
	bCyclePause					: BOOL;			(* Cr800 cycle is stopping *)
	bRestoreAuto				: BOOL;			(* CR800 is restoring auto mode *)
	bRestoreCycle				: BOOL;			(* CR800 is restoring cycle *)
	iActionNumber				: UINT;
	bAbort						: BOOL;			(* Deinitialize function block *)
	bError		 				: BOOL;			(* FB error occuring*)
	bDontSetInitialParameters	: BOOL;			(* Don't set initial parameters in initalization *)
	bBusy						: BOOL;
	bActive						: BOOL;
	bAutoModeStarted			: BOOL;
	bUninitialized				: BOOL; 
	bStopped					: BOOL;
	bInitProgram				: BOOL;
	bSendPosition1				: BOOL;
	bSendPosition2				: BOOL;
	bGetPosition				: BOOL;
	
	eErrorID 					: E_CR800Error;	(*  *)
	
	eCR800State					: E_CR800State					:= 0; (* Main state machine of function block *)
	eCR800StateBeforeReset		: E_CR800State					:= 0; (* State of CR800 before reseting the error *)
	eCR800StateHome 			: E_CR800StateHoming 			:= 0; (* State machine of homing *)
	eCR800StateDoRequest		: E_CR800StateDoingRequest		:= 0; (* State machine of executing request*)
	eCR800StateReceiveCommand	: E_CR800StateCommandExchange	:= 0; (* State machine of receive command data exchange *) 
	eCR800SendCommand			: E_CR800StateCommandExchange	:= 0; (* State machine of send commad data exchange *) 
	eCR800StateAbort 			: E_CR800StateAborting 			:= 0; (* State machine of aboriting *) 
	eCR800StateInitializing 	: E_CR800StateInitializing 		:= 0; (* State machine of initilaizing *)
	eCR800StateCycleStop 		: E_CR800StateCycleStopping		:= 0; (* State machine of cycle stopping *)
	eCR800StateCyclePause		: E_CR800StateCyclePausing		:= 0; (* State machine of cycle Pausing *)
	eCR800StateBeforeSendPosition : E_CR800State				:= 0;
	eCR800StateSendPosition		: E_CR800StateSendPosition		:= 0; (* State machine of cycle Pausing *)

	stRobot						: ST_VisuCtrlRobotFrame; 
	
	iOverride					: USINT;
	lrPositionX1				: LREAL;
	lrPositionY1				: LREAL;
	lrRotation1					: LREAL;
	lrPositionX2				: LREAL;
	lrPositionY2				: LREAL;
	lrRotation2					: LREAL;
	
	stUserDefinedArea			: ST_CR800UserDefinedArea;
	
	(* Timers *)
	tTimeout					: TIME := tWATCHDOG_TIMEOUT;	(**)
	tonWatchdog					: TON;							(* Input timeout watchdog *)

	feTrigStopped 				: F_TRIG;
	//rtErrorOccuring				: R_TRIG;
END_VAR

M_ConvertEthercatData() ;

//rtErrorOccuring(CLK := ErrorOccuring);
IF ErrorOccuring THEN
	//rtErrorOccuring(CLK := FALSE);
	eCR800State := CR800_IN_EXTERNAL_ERROR ;
	bError := TRUE ;
	eErrorID := CR800_ERROR_CR800_ERROR_OCCURING ;
END_IF

ActionNumber := iActionNumber;
stCR800EthercatData.arrRegistersOutput[6021] := USINT_TO_INT(iOverride);

StateMachine() ;

feTrigStopped(CLK := CycleStopping);

IF feTrigStopped.Q THEN 
	bStopped := TRUE;
END_IF

tonWatchdog(PT := tTimeout) ;

//stCR800EthercatData.arrRegistersOutput[6021] := 100 ; {warning 'Odhardkodować - przenieść do receptury'}

PROPERTY ActionNumber : UINT
GET
ActionNumber := iActionNumber;
END_GET
SET
IF ActionNumber >= 13 AND ActionNumber <= 100 THEN
	iActionNumber := ActionNumber;
END_IF
END_SET
END_PROPERTY

PROPERTY Active : REFERENCE TO BOOL
GET
Active REF= bActive;
END_GET
END_PROPERTY

PROPERTY AutoModeStarted : REFERENCE TO BOOL
GET
AutoModeStarted REF= bAutoModeStarted;
END_GET
END_PROPERTY

(* Desription from CR800 side:
"Outputs that the controller battery voltage is
low. The output is turned off when the
controller power supply is reconnected after
the battery replacement.
*The cumulative time where the controller
power supply is turned off exceeds 14600
hours.
The output is turned off if the battery depletion
time is reset." *)
{attribute 'monitoring' := 'variable'}
PROPERTY PUBLIC BatteryLow : BOOL ;
GET
BatteryLow := stCR800EthercatData.arrSignalsInputConverted[6014] ;
END_GET
END_PROPERTY

(* Desription from CR800 side:
Reset the battery cumulative tine. *) 
{attribute 'monitoring' := 'variable'}
PROPERTY BatteryReset : BOOL
GET
BatteryReset := stCR800EthercatData.arrSignalsOutputConverted[6015] ;
END_GET
SET
stCR800EthercatData.arrSignalsOutputConverted[6015] := BatteryReset ;
END_SET
END_PROPERTY

(* Desription from a CR800 side:
Output that the reset has been completed *)
{attribute 'monitoring' := 'variable'}
PROPERTY PUBLIC BatteryResetCompleted : BOOL ;
GET
BatteryResetCompleted := stCR800EthercatData.arrSignalsInputConverted[6015] ;
END_GET
END_PROPERTY

PROPERTY Busy : REFERENCE TO BOOL
GET
Busy REF= bBusy;
END_GET
END_PROPERTY

(* Desription from CR800 side:
Outputs that the power has been turned ON
and that the external input signal can be
received *)
{attribute 'monitoring' := 'variable'}
PROPERTY PUBLIC CR800PoweredOn : BOOL ;
GET
CR800PoweredOn := stCR800EthercatData.arrSignalsInputConverted[6000] ;
END_GET
END_PROPERTY

(* Desription from a CR800 side:
Starts the cycle stop *)
{attribute 'monitoring' := 'variable'}
PROPERTY CycleStop : BOOL
GET
CycleStop := stCR800EthercatData.arrSignalsOutputConverted[6013] ;
END_GET
SET
stCR800EthercatData.arrSignalsOutputConverted[6013] := CycleStop;
END_SET
END_PROPERTY

(* Desription from CR800 side:
"Outputs that the cycle stop is operating.
Turns OFF when the cycle stop is completed" *)
{attribute 'monitoring' := 'variable'}
PROPERTY PUBLIC CycleStopping : BOOL ;
GET
CycleStopping := stCR800EthercatData.arrSignalsInputConverted[6013] ;
END_GET
END_PROPERTY

PROPERTY DoingAction : REFERENCE TO BOOL
GET
DoingAction REF= bDoAction;
END_GET
END_PROPERTY

(*Desription from a CR800 side:
"Outputs that an emergency stop is occurring.
[EMGERR output conditions]
• External emergency stop error:
H0050, H0051 (Dual line is faulty)
• Operation panel emergency stop error:
H0060, H0061 (Dual line is faulty)
• T/B emergency stop error:
H0070, H0071 (Dual line is faulty)
• Door switch signal faulty:
H0039, H0040 (Dual line is faulty)
• Wiring error of EMG connector:
H0141"*)
{attribute 'monitoring' := 'variable'}
PROPERTY PUBLIC EmergencyStopOccuring : BOOL ;
GET
EmergencyStopOccuring := stCR800EthercatData.arrSignalsInputConverted[6016] ;
END_GET
END_PROPERTY

PROPERTY Error : REFERENCE TO BOOL
GET
Error REF= bError;
END_GET
END_PROPERTY

(* Actual FB error *)
{attribute 'monitoring' := 'variable'}
PROPERTY Errorname : STRING
GET
Errorname := TO_STRING(eErrorID) ;
END_GET
END_PROPERTY

{attribute 'monitoring' := 'variable'}
PROPERTY PUBLIC ErrorOccuring : BOOL ;
(*Desription from CR800 side:
Outputs that an error has occurred.
*)
GET
ErrorOccuring := stCR800EthercatData.arrSignalsInputConverted[6010] ;
END_GET
END_PROPERTY

(* Desription from CR800 side:
This input stops the program being executed.
(The specification is the same as for the STOP
parameter.)
Unlike the STOP parameter, signal numbers
can be changed. *)
{attribute 'monitoring' := 'variable'}
PROPERTY ErrorReset : BOOL
GET
ErrorReset := stCR800EthercatData.arrSignalsOutputConverted[6010] ;
END_GET
SET
stCR800EthercatData.arrSignalsOutputConverted[6010] := ErrorReset ;
END_SET
END_PROPERTY

PROPERTY EthercatData : REFERENCE TO ST_CR800EthercatData
GET
EthercatData REF= stCR800EthercatData;
END_GET
END_PROPERTY

(*Desription from CR800 side:
This output indicates that the controller mode
is set to AUTOMATIC.*)
{attribute 'monitoring' := 'variable'}
PROPERTY PUBLIC InAutomaticMode : BOOL ;
GET
InAutomaticMode := stCR800EthercatData.arrSignalsInputConverted[6003] ;
END_GET
END_PROPERTY

(* Desription from CR800 side:
This output indicates that the controller mode
is set to AUTOMATIC and remote operation
mode.*)
{attribute 'monitoring' := 'variable'}
PROPERTY PUBLIC InRemoteMode : BOOL ;
GET
InRemoteMode := stCR800EthercatData.arrSignalsInputConverted[6001] ;
END_GET
END_PROPERTY

(*Desription from CR800 side:
This output indicates that the controller mode
is set to Teaching mode. *)
{attribute 'monitoring' := 'variable'}
PROPERTY PUBLIC InTeachingMode : BOOL ;
GET
InTeachingMode := stCR800EthercatData.arrSignalsInputConverted[6002] ;
END_GET
END_PROPERTY

PROPERTY IsHomed : REFERENCE TO BOOL
GET
IsHomed REF= bIsHomed;
END_GET
END_PROPERTY

(*This mehtod converts raw data from memory and converts its number for the same like in the mitshubishi manual
  F:\Dept\SMT\Electronics\Mitsubishi\Manuals\Karta ethercat*)
METHOD Protected M_ConvertEthercatData : BOOL
VAR
	iLoop	: INT;	
END_VAR
FOR iLoop := 0 TO 31 DO  
	stCR800EthercatData.arrSignalsInputConverted[iMIN_ETHERCAT_REGISTER_IN_CR800  +iLoop*8]	:= 	stCR800EthercatData.arrSignalsInputRaw[iLoop].0	;
	stCR800EthercatData.arrSignalsInputConverted[iMIN_ETHERCAT_REGISTER_IN_CR800+1+iLoop*8]	:= 	stCR800EthercatData.arrSignalsInputRaw[iLoop].1	;
	stCR800EthercatData.arrSignalsInputConverted[iMIN_ETHERCAT_REGISTER_IN_CR800+2+iLoop*8] := 	stCR800EthercatData.arrSignalsInputRaw[iLoop].2	;
	stCR800EthercatData.arrSignalsInputConverted[iMIN_ETHERCAT_REGISTER_IN_CR800+3+iLoop*8] := 	stCR800EthercatData.arrSignalsInputRaw[iLoop].3	;
	stCR800EthercatData.arrSignalsInputConverted[iMIN_ETHERCAT_REGISTER_IN_CR800+4+iLoop*8] := 	stCR800EthercatData.arrSignalsInputRaw[iLoop].4	;
	stCR800EthercatData.arrSignalsInputConverted[iMIN_ETHERCAT_REGISTER_IN_CR800+5+iLoop*8] := 	stCR800EthercatData.arrSignalsInputRaw[iLoop].5	;
	stCR800EthercatData.arrSignalsInputConverted[iMIN_ETHERCAT_REGISTER_IN_CR800+6+iLoop*8] := 	stCR800EthercatData.arrSignalsInputRaw[iLoop].6	;
	stCR800EthercatData.arrSignalsInputConverted[iMIN_ETHERCAT_REGISTER_IN_CR800+7+iLoop*8] := 	stCR800EthercatData.arrSignalsInputRaw[iLoop].7	;
	
	stCR800EthercatData.arrSignalsOutputRaw[iLoop].0	:=	stCR800EthercatData.arrSignalsOutputConverted[iMIN_ETHERCAT_REGISTER_IN_CR800  +iLoop*8];
	stCR800EthercatData.arrSignalsOutputRaw[iLoop].1	:=	stCR800EthercatData.arrSignalsOutputConverted[iMIN_ETHERCAT_REGISTER_IN_CR800+1+iLoop*8];
	stCR800EthercatData.arrSignalsOutputRaw[iLoop].2	:=	stCR800EthercatData.arrSignalsOutputConverted[iMIN_ETHERCAT_REGISTER_IN_CR800+2+iLoop*8];
	stCR800EthercatData.arrSignalsOutputRaw[iLoop].3	:=	stCR800EthercatData.arrSignalsOutputConverted[iMIN_ETHERCAT_REGISTER_IN_CR800+3+iLoop*8];
	stCR800EthercatData.arrSignalsOutputRaw[iLoop].4	:=	stCR800EthercatData.arrSignalsOutputConverted[iMIN_ETHERCAT_REGISTER_IN_CR800+4+iLoop*8];
	stCR800EthercatData.arrSignalsOutputRaw[iLoop].5	:=	stCR800EthercatData.arrSignalsOutputConverted[iMIN_ETHERCAT_REGISTER_IN_CR800+5+iLoop*8];
	stCR800EthercatData.arrSignalsOutputRaw[iLoop].6	:=	stCR800EthercatData.arrSignalsOutputConverted[iMIN_ETHERCAT_REGISTER_IN_CR800+6+iLoop*8];
	stCR800EthercatData.arrSignalsOutputRaw[iLoop].7	:=	stCR800EthercatData.arrSignalsOutputConverted[iMIN_ETHERCAT_REGISTER_IN_CR800+7+iLoop*8];
END_FOR
END_METHOD

(* 1 - Request executed, 0 - request not executed 
	Description:
		This method doing request robot to do request with given number in iNumberOfRequest *)

METHOD PROTECTED M_DoRequest : BOOL
VAR_INPUT
	iNumberOfRequest	: 	UINT	;	(* Destination memory place in the robot*)
END_VAR
CASE eCR800StateDoRequest OF

	CR800_DOING_REQUEST_IDLE:
		M_DoRequest			:= FALSE ;
		eCR800StateDoRequest		:= CR800_DOING_REQUEST_SEND_REQUEST;
		
	CR800_DOING_REQUEST_SEND_REQUEST:
		IF M_SendCommand(iDestinationAdress := iSEND_REQUEST_ADDRESS, iRequestNumber := iNumberOfRequest) THEN
			eCR800StateDoRequest	:= CR800_DOING_REQUEST_WAIT_FOR_CONFIRM;
		END_IF
		
	CR800_DOING_REQUEST_WAIT_FOR_CONFIRM:
		IF M_ReceiveCommand(iDestinationAdress := iRECEIVE_REQUEST_ADDRESS) THEN
			eCR800StateDoRequest 	:= CR800_DOING_REQUEST_DONE ;
		END_IF
	
	CR800_DOING_REQUEST_DONE:
		M_DoRequest			:= TRUE ;
		eCR800StateDoRequest 		:= CR800_DOING_REQUEST_IDLE ;
END_CASE
END_METHOD

(*1 - Operation rights granted, 0 - Operation rights not granted
	Description: 
		This method grants operation rights to the PLC in CR800
		IE. PLC is only controlling the robot.
		Warning: The operation rights is lost, when teaching box is in the "Operation panel" screen.
		Input bRequest: 1 - Enable, 0 - unable *) 

METHOD PROTECTED M_OperationRigtsEnable : BOOL 
VAR_INPUT
	bRequest : BOOL ; (*1 - Enable, 0 - unable *) 
END_VAR
IF bRequest THEN 
	OperationRightsEnable := TRUE ;
	tonWatchdog.IN := TRUE ;
	IF OperationRightsEnabled THEN
		tonWatchdog.IN := FALSE ;
		M_OperationRigtsEnable := TRUE ;
	//ELSIF tonWatchdog.Q THEN
	//	bError 		:= TRUE ;
	//	eErrorID	:= CR800_ERROR_GRANTING_OPERATION_RIGHTS_TIMED_OUT ;			
	END_IF
END_IF

IF NOT bRequest THEN 
	OperationRightsEnable := FALSE ;
	tonWatchdog.IN := TRUE ;
	IF NOT OperationRightsEnabled THEN
		tonWatchdog.IN := FALSE ;
		M_OperationRigtsEnable := FALSE ;
	ELSIF tonWatchdog.Q THEN
		bError 		:= TRUE ;
		eErrorID	:= CR800_ERROR_ABORTING_OPERATION_RIGHTS_TIMED_OUT ;			
	END_IF
END_IF
END_METHOD

(* 1 - Program is reseted, 0 - program is not reseted
	Description:
		This method reset the program in Cr800
		IE. The next program start will begin form the first line*)
METHOD PROTECTED M_ProgramReset : BOOL
VAR_INPUT
END_VAR
IF ProgramOperating THEN
	bError 		:= TRUE ;
	eErrorID	:= CR800_ERROR_CANT_RESET_PRG_DURING_PRG_RUN ;
ELSE
	ProgramReset 	:= TRUE	;
	tonWatchdog.IN 	:= TRUE ;
	IF ProgramSelectionEnabled THEN
		ProgramReset 	:= FALSE;
		tonWatchdog.IN 	:= FALSE;	
		M_ProgramReset := TRUE ;
	ELSIF tonWatchdog.Q THEN
		bError 			:= TRUE ;
		eErrorID		:= CR800_ERROR_RESET_PRG_TIMED_OUT ;			
	END_IF
END_IF
END_METHOD

(* 0 - program not started, 1 - Program started 
	Description:
		This method starts the program in CR800 *) 
METHOD protected M_ProgramStart : BOOL
IF tonWatchdog.Q THEN
	bError 			:= TRUE ;
	eErrorID		:= CR800_ERROR_START_PRG_TIMED_OUT ;	
ELSIF NOT ProgramOperating OR StopSTS THEN
	ProgramStart 	:= TRUE	;
	M_ProgramStart := FALSE;
	tonWatchdog.IN 	:= TRUE ;
ELSIF ProgramOperating THEN
	ProgramStart 	:= FALSE;
	M_ProgramStart := TRUE ;
	tonWatchdog.IN 	:= FALSE;		
END_IF
END_METHOD

(* 1 - program stopped, 0 - program has not stopped
	Description:
		This method stops (pause) the program in CR800.
		IE. Stops the program implicitly *)
METHOD PROTECTED  M_ProgramStop : BOOL
M_ProgramStop  := FALSE ;
ProgramStop2 	:= TRUE ;

IF StopSTS AND NOT ProgramOperating THEN
	ProgramStop2	:= FALSE ;
	M_ProgramStop  := TRUE ;
END_IF
END_METHOD

(* 0 - command not Received, 1 - command Received 
	Desription:
		This method waits for the information from the iDestinationAddress, send confirmation,
 		waits for reset command and then resets confirmation *)
{attribute 'monitoring' := 'variable'}
METHOD PROTECTED M_ReceiveCommand : BOOL 
VAR_INPUT
	iDestinationAdress	: 	UINT	;	(* Destination memory place in the robot*)
END_VAR
//IF tonWatchdog.Q THEN
//	bError 		:= TRUE ;
//	eErrorID	:= CR800_ERROR_RECEIVE_COMMAND_TIMED_OUT ;			
//END_IF

CASE eCR800StateReceiveCommand OF
	
	CR800_CMD_EXCHANGE_IDLE:
		M_ReceiveCommand := FALSE ;
//		tonWatchdog.IN 	:= TRUE ;
		eCR800StateReceiveCommand 	:= CR800_CMD_EXCHANGE_WAIT_FOR_DATA ;

	CR800_CMD_EXCHANGE_WAIT_FOR_DATA:
		IF stCR800EthercatData.arrSignalsInputConverted[iDestinationAdress] THEN
			eCR800StateReceiveCommand := CR800_CMD_EXCHANGE_SEND_CONFIRMATION ;			
		END_IF

	CR800_CMD_EXCHANGE_SEND_CONFIRMATION:
		stCR800EthercatData.arrSignalsOutputConverted[iDestinationAdress] := TRUE ;
		eCR800StateReceiveCommand 	:= CR800_CMD_EXCHANGE_WAIT_FOR_RESET_COMMAND ;
		
	CR800_CMD_EXCHANGE_WAIT_FOR_RESET_COMMAND:
		IF NOT stCR800EthercatData.arrSignalsInputConverted[iDestinationAdress] THEN
			eCR800StateReceiveCommand := CR800_CMD_EXCHANGE_RESET_ITERLOCKS ;			
		END_IF
			
	CR800_CMD_EXCHANGE_RESET_ITERLOCKS:
		stCR800EthercatData.arrSignalsOutputConverted[iDestinationAdress] := FALSE;
		eCR800StateReceiveCommand	:= CR800_CMD_EXCHANGE_DONE ;

	CR800_CMD_EXCHANGE_DONE:
//		tonWatchdog.IN 					:= FALSE;	
		M_ReceiveCommand 				:= TRUE ;		
		eCR800StateReceiveCommand	:= CR800_CMD_EXCHANGE_IDLE ;

END_CASE
END_METHOD

(* Desription:
	This method resets fb variables *)
METHOD PROTECTED M_ResetVariables : BOOL
VAR
	iLoop: INT;
END_VAR
//M_OperationRigtsEnable(bRequest 	:= 0);
eCR800StateDoRequest				:= 0 ;
eCR800StateHome 					:= 0 ;	
eCR800StateReceiveCommand			:= 0 ;
eCR800SendCommand					:= 0 ;
eCR800StateInitializing 			:= 0 ;
eCR800StateCycleStop 				:= 0 ; 
eCR800StateCyclePause				:= 0 ; 
eCR800StateSendPosition				:= 0 ;

eErrorID := CR800_ERROR_OK;

bGoHome 			:=	FALSE;
bUpdateRecipes		:=	FALSE;
bGoAuto				:=	FALSE;
bDoAction			:=	FALSE;
bCycleStop			:=	FALSE;
bCyclePause			:= 	FALSE;
bRestoreCycle		:=  FALSE;
bIsHomed			:=	FALSE;
bAutoModeStarted 	:=  FALSE;
tonWatchdog.IN 		:=  FALSE;

FOR iLoop := iMIN_ETHERCAT_REGISTER_IN_CR800 TO iMAX_ETHERCAT_REGISTER_IN_CR800 DO
	stCR800EthercatData.arrRegistersOutput[iLoop] 			:= 0 ;
	stCR800EthercatData.arrSignalsOutputConverted[iLoop]	:= 0 ;
END_FOR
END_METHOD

(* 0 - command not sent, 1 - command sent 
	Descritpion:
		This method sends the information to the iDestinationAddress, waits for a confirmation,
 		send reset command and then resets send request *)
{attribute 'monitoring' := 'variable'}
METHOD PROTECTED M_SendCommand : BOOL

VAR_INPUT
	iDestinationAdress		: 	UINT	;	(* Destination memory place in the robot*)
	iRequestNumber			:  	UINT	;	(* Reqest number that robot has to perform *)		
END_VAR
IF tonWatchdog.Q THEN
	bError 		:= TRUE ;
	eErrorID	:= CR800_ERROR_SEND_COMMAND_TIMED_OUT ;			
END_IF


CASE eCR800SendCommand OF
	
	CR800_CMD_EXCHANGE_IDLE:
		M_SendCommand 	:= FALSE ;
		RequestNumber 	:= iRequestNumber ; 
		tonWatchdog.IN 	:= TRUE ;
		eCR800SendCommand 	:= CR800_CMD_EXCHANGE_SEND_DATA ;

	CR800_CMD_EXCHANGE_SEND_DATA:
		stCR800EthercatData.arrSignalsOutputConverted[iDestinationAdress] := TRUE ;
		eCR800SendCommand 	:= CR800_CMD_EXCHANGE_WAIT_FOR_CONFIRMATION ;
		
	CR800_CMD_EXCHANGE_WAIT_FOR_CONFIRMATION:
		IF stCR800EthercatData.arrSignalsInputConverted[iDestinationAdress] THEN
			eCR800SendCommand := CR800_CMD_EXCHANGE_RESET_ITERLOCKS ;			
		END_IF
	
	CR800_CMD_EXCHANGE_RESET_ITERLOCKS:
		stCR800EthercatData.arrSignalsOutputConverted[iDestinationAdress] := FALSE;
		eCR800SendCommand	:= CR800_CMD_EXCHANGE_WAIT_FOR_RESET_CONFIRMATION ;
	
	CR800_CMD_EXCHANGE_WAIT_FOR_RESET_CONFIRMATION:
		IF NOT stCR800EthercatData.arrSignalsInputConverted[iDestinationAdress] THEN
			eCR800SendCommand := CR800_CMD_EXCHANGE_DONE ;			
		END_IF
		
	CR800_CMD_EXCHANGE_DONE:
		tonWatchdog.IN 				:= FALSE;
		M_SendCommand 				:= TRUE ;
		eCR800SendCommand 	:= CR800_CMD_EXCHANGE_IDLE ;
END_CASE
END_METHOD

(* Servo Off request. 1 - Servo offed succesfully, 0 - Servo has not stopped yet
	Description:
		This method turns off the servos of the robot *)
METHOD PROTECTED M_ServoOff : BOOL
ServoOFF := TRUE ;

IF ServoIsOff THEN
	ServoOFF 	:= FALSE ;
	M_ServoOFF := TRUE ;
END_IF
END_METHOD

(* 1 - Servo on succesfully, 0 - Servo has not stopped yet
	Description:
		This method turns on the servos of the robot *)
METHOD PROTECTED M_ServoOn : BOOL (*Servo ON request*)
IF NOT ServoOFF THEN

	ServoON 		:= TRUE ;
	tonWatchdog.IN 	:= TRUE ;
	IF ServoIsOn THEN
		ServoON 		:= FALSE ;
		M_ServoON 		:= TRUE	 ;
		tonWatchdog.IN 	:= FALSE ;
	ELSIF tonWatchdog.Q THEN
		bError 		:= TRUE ;
		eErrorID	:= CR800_ERROR_SERVO_ON_TIMED_OUT ;			
	END_IF
	
END_IF
END_METHOD

(* Actual state of main state machine *)
{attribute 'monitoring' := 'variable'}
PROPERTY MainStateMachine : STRING
GET
MainStateMachine := TO_STRING(eCR800State) ;
END_GET
END_PROPERTY

(* 1 - abroting finished, 0 - aborting not finished.
	Description:
		This method aborts all actions, stops and reset the program and turn off the robot*)
METHOD  MR_Abort : BOOL
IF eCR800State <> CR800_UNINITIALIZED OR ServoIsOn THEN
	bBusy 	:= TRUE;
	bAbort := TRUE;
	MR_Abort := FALSE;
	eCR800State := CR800_ABORTING;
	fbMachineLogger.MR_AddLogs(CONCAT(sName,' : abort requested'));	
	
ELSIF eCR800State = CR800_UNINITIALIZED THEN
	bAbort := FALSE;
	MR_Abort := TRUE;
//	bActive := FALSE; 
	bBusy 	:= FALSE;
	fbMachineLogger.MR_AddLogs(CONCAT(sName,' : abort done'));	
	
END_IF
END_METHOD

